// EVENT CODE //
	FB_AlarmCodeManager(
		bAlarm1			:= TON_BatteriesCharging.Q ,								//Batteries charging
		bAlarm2			:= TON_BatteriesDischarging.Q,								//Batteries discharging
		bAlarm3			:= FALSE,													//
		bAlarm4			:= FALSE,													//		
		bAlarm5			:= IN_CmdOpenDC,                                            // Open DC command
		bAlarm6			:= IN_CmdCloseDC,                                           // Close DC Command
		bAlarm7			:= FALSE,                                                   //
		bAlarm8			:= FALSE,                                                   //
		bAlarm9			:= FALSE,                                                   //
		bAlarm10		:= FALSE,                                                   //
		bAlarm11		:= FALSE,                                                   //
		bAlarm12		:= FALSE,                                                   //
		bAlarm13		:= FALSE,                                                   //
		bAlarm14		:= FALSE,                                                   //
		bAlarm15		:= FALSE,                                                   //
		wAlarmCode		=> MesDataExd.MesData.MesEventCode);


	FB_AlarmCodeManager(	
        bAlarm1			:= MesDataExd.MesChargeStatus= 1,  									// Charge Status  -  OFF
        bAlarm2			:= MesDataExd.MesChargeStatus= 2,  									// Charge Status  -  EMPTY
        bAlarm3			:= MesDataExd.MesChargeStatus= 3,  									// Charge Status  -  DISCHARGING
        bAlarm4			:= MesDataExd.MesChargeStatus= 4,  									// Charge Status  -  CHARGING
        bAlarm5			:= MesDataExd.MesChargeStatus= 5,  									// Charge Status  -  FULL
        bAlarm6			:= MesDataExd.MesChargeStatus= 6,  									// Charge Status  -  HOLDING
        bAlarm7			:= MesDataExd.MesChargeStatus= 7,  									// Charge Status  -  TESTING
		bAlarm8			:= FALSE,                                                   //
		bAlarm9			:= FALSE,                                                   //
		bAlarm10		:= FALSE,                                                   //
		bAlarm11		:= FALSE,                                                   //
		bAlarm12		:= FALSE,                                                   //
		bAlarm13		:= FALSE,                                                   //
		bAlarm14		:= FALSE,                                                   //
		bAlarm15		:= FALSE,                                                   //
		wAlarmCode		=> MesDataExd.MesChargeStatus);

		

	FB_AlarmCodeManager(	
        bAlarm1			:= MesIDState= 1,  				// State of the Battery Bank  -  DISCONNECTED
        bAlarm2			:= MesIDState= 2,  				// State of the Battery Bank  -  INITIALIZING
        bAlarm3			:= MesIDState= 3,  				// State of the Battery Bank  -  CONNECTED
        bAlarm4			:= MesIDState= 4,  				// State of the Battery Bank  -  STANDBY
        bAlarm5			:= MesIDState= 5,  				// State of the Battery Bank  -  SOC PROTECTION
        bAlarm6			:= MesIDState= 6,  				// State of the Battery Bank  -  SUSPENDING
        bAlarm7			:= MesIDState= 99,  			// State of the Battery Bank  -  FAULT
		bAlarm8			:= FALSE,                       //
		bAlarm9			:= FALSE,                       //
		bAlarm10		:= FALSE,                       //
		bAlarm11		:= FALSE,                       //
		bAlarm12		:= FALSE,                       //
		bAlarm13		:= FALSE,                       //
		bAlarm14		:= FALSE,                       //
		bAlarm15		:= FALSE,                       //
		wAlarmCode		=> MesDataExd.MesData.MesIDState
);
(*
	FB_AlarmCodeManager(	
        bAlarm1		:= MesData.MesEvt1.0,  			// Battery Event 1 -  COMMUNICATION_ERROR
        bAlarm2		:= MesData.MesEvt1.1,  			// Battery Event 1 -  OVER_TEMP_ALARM
        bAlarm3		:= MesData.MesEvt1.2,  			// Battery Event 1 -  OVER_TEMP_WARNING
        bAlarm4		:= MesData.MesEvt1.3,  			// Battery Event 1 -  UNDER_TEMP_ALARM
        bAlarm5		:= MesData.MesEvt1.4,  			// Battery Event 1 -  UNDER_TEMP_WARNING
        bAlarm6		:= MesData.MesEvt1.5,  			// Battery Event 1 -  OVER_CHARGE_CURRENT_ALARM
        bAlarm7		:= MesData.MesEvt1.6,  			// Battery Event 1 -  OVER_CHARGE_CURRENT_WARNING
        bAlarm8		:= MesData.MesEvt1.7,  			// Battery Event 1 -  OVER_DISCHARGE_CURRENT_ALARM
        bAlarm9		:= MesData.MesEvt1.8,  			// Battery Event 1 -  OVER_DISCHARGE_CURRENT_WARNING
        bAlarm10	:= MesData.MesEvt1.9,  			// Battery Event 1 -  OVER_VOLT_ALARM
        bAlarm11	:= MesData.MesEvt1.10,  		// Battery Event 1 -  OVER_VOLT_WARNING
        bAlarm12	:= MesData.MesEvt1.11,  		// Battery Event 1 -  UNDER_VOLT_ALARM
        bAlarm13	:= MesData.MesEvt1.12,  		// Battery Event 1 -  UNDER_VOLT_WARNING
        bAlarm14	:= MesData.MesEvt1.13,  		// Battery Event 1 -  UNDER_SOC_MIN_ALARM
        bAlarm15	:= MesData.MesEvt1.14,  		// Battery Event 1 -  UNDER_SOC_MIN_WARNING
		wAlarmCode	=> MesData.MesAlarmCode_MesEvt1_1
);

	FB_AlarmCodeManager(	
        bAlarm1		:= MesData.MesEvt1.15,  		// Battery Event 1 -  OVER_SOC_MAX_ALARM
        bAlarm2		:= MesData.MesEvt1.16,  		// Battery Event 1 -  OVER_SOC_MAX_WARNING
        bAlarm3		:= MesData.MesEvt1.17,  		// Battery Event 1 -  VOLTAGE_IMBALANCE_WARNING
        bAlarm4		:= MesData.MesEvt1.18,  		// Battery Event 1 -  TEMPERATURE_IMBALANCE_ALARM
        bAlarm5		:= MesData.MesEvt1.19,  		// Battery Event 1 -  TEMPERATURE_IMBALANCE_WARNING
        bAlarm6		:= MesData.MesEvt1.20,  		// Battery Event 1 -  CONTACTOR_ERROR
        bAlarm7		:= MesData.MesEvt1.21,  		// Battery Event 1 -  FAN_ERROR
        bAlarm8		:= MesData.MesEvt1.22,  		// Battery Event 1 -  GROUND_FAULT
        bAlarm9		:= MesData.MesEvt1.23,  		// Battery Event 1 -  OPEN_DOOR_ERROR
        bAlarm10	:= MesData.MesEvt1.24,  		// Battery Event 1 -  CURRENT_IMBALANCE_WARNING
        bAlarm11	:= MesData.MesEvt1.25,  		// Battery Event 1 -  OTHER_ALARM
        bAlarm12	:= MesData.MesEvt1.26,  		// Battery Event 1 -  OTHER_WARNING
        bAlarm13	:= MesData.MesEvt1.27,  		// Battery Event 1 -  RESERVED_1
        bAlarm14	:= MesData.MesEvt1.28,  		// Battery Event 1 -  CONFIGURATION_ALARM
        bAlarm15	:= MesData.MesEvt1.29,  		// Battery Event 1 -  CONFIGURATION_WARNING
		wAlarmCode	=> MesData.MesAlarmCode_MesEvt1_2
);

	FB_AlarmCodeManager(	
        bAlarm1			:= MesData.MesEvtVnd1.0,  		// Battery Vendor Event 1   -  Cell Over Voltage Warning   
        bAlarm2			:= MesData.MesEvtVnd1.1,  		// Battery Vendor Event 1   -  Cell Under Voltage Warning  
        bAlarm3			:= MesData.MesEvtVnd1.2,  		// Battery Vendor Event 1   -  Cell Voltage Imbalance      
        bAlarm4			:= MesData.MesEvtVnd1.3,  		// Battery Vendor Event 1   -  Cell Over Voltage Alarm     
        bAlarm5			:= MesData.MesEvtVnd1.4,  		// Battery Vendor Event 1   -  Cell Under Voltage Alarm    
        bAlarm6			:= MesData.MesEvtVnd1.5,  		// Battery Vendor Event 1   -  Cell Voltage Imbalance Alarm
        bAlarm7			:= MesData.MesEvtVnd1.6,  		// Battery Vendor Event 1   -  Cell Over Voltage Fault     
        bAlarm8			:= MesData.MesEvtVnd1.7,  		// Battery Vendor Event 1   -  Cell Under Voltage Fault    
        bAlarm9			:= MesData.MesEvtVnd1.8,  		// Battery Vendor Event 1   -  Cell Voltage Imbalance Fault
        bAlarm10		:= MesData.MesEvtVnd1.9,  		// Battery Vendor Event 1   -  Over Temperature Fault      
        bAlarm11		:= MesData.MesEvtVnd1.10,  	// Battery Vendor Event 1   -  Under Temperature Fault     
        bAlarm12		:= MesData.MesEvtVnd1.11,  	// Battery Vendor Event 1   -  Temperature Imbalance Fault 
        bAlarm13		:= MesData.MesEvtVnd1.12,  	// Battery Vendor Event 1   -  Over Voltage Fault          
        bAlarm14		:= MesData.MesEvtVnd1.13,  	// Battery Vendor Event 1   -  Under Voltage Fault         
        bAlarm15		:= MesData.MesEvtVnd1.14,  	// Battery Vendor Event 1   -  Over Charge Current Fault   
		wAlarmCode		=>MesData.MesAlarmCode_MesEvtVnd1_1
);

	FB_AlarmCodeManager(	
        bAlarm1			:= MesData.MesEvtVnd1.15,  	// Battery Vendor Event 1  -  Over Discharge Current Fault      
        bAlarm2			:= MesData.MesEvtVnd1.16,  	// Battery Vendor Event 1  -  String Connection Failure         
        bAlarm3			:= MesData.MesEvtVnd1.17,  	// Battery Vendor Event 1  -  RBMS to MBMS Communication Failure
        bAlarm4			:= MesData.MesEvtVnd1.18,  	// Battery Vendor Event 1  -  Temperature Sensor Failure       
        bAlarm5			:= MesData.MesEvtVnd1.19,  	// Battery Vendor Event 1  -  Main Relay Open Failure          
        bAlarm6			:= MesData.MesEvtVnd1.20,  	// Battery Vendor Event 1  -  Bus Voltage Imbalance             
        bAlarm7			:= MesData.MesEvtVnd1.21,  	// Battery Vendor Event 1  -  Fan Failure                       
        bAlarm8			:= MesData.MesEvtVnd1.22,  	// Battery Vendor Event 1  -  Voltage Sensor Failure            
        bAlarm9			:= MesData.MesEvtVnd1.23,  	// Battery Vendor Event 1  -  Insulation Detection Warning      
        bAlarm10		:= MesData.MesEvtVnd1.24,  	// Battery Vendor Event 1  -  Insulation Detection Fault        
		bAlarm11		:= FALSE,                                                   //
		bAlarm12		:= FALSE,                                                   //
		bAlarm13		:= FALSE,                                                   //
		bAlarm14		:= FALSE,                                                   //
		bAlarm15		:= FALSE,                                                   //
		wAlarmCode		=> MesData.MesAlarmCode_MesEvtVnd1_2
);
*)
END_METHOD

METHOD M_CP
//////////////////
//  Permanent conditions 
/////////////////

VAR 
	// Method local variables (reinitialized at each cycle) 
	
END_VAR


SUPER^.M_CP() ; 




Trig_Cmd_Read(CLK:=IN_CmdToggleRead);
Trig_Cmd_Write(CLK:=IN_CmdToggleWrite);
	
IF Trig_Cmd_Read.Q THEN
	IN_CmdToggleRead := FALSE;
	MesDataExd.MesData.MesCP_Read := NOT MesDataExd.MesData.MesCP_Read;
END_IF


IF Trig_Cmd_Write.Q THEN
	IN_CmdToggleWrite := FALSE;
	MesDataExd.MesData.MesCP_Write := NOT MesDataExd.MesData.MesCP_Write;
END_IF
END_METHOD

METHOD M_Evaluate : BOOL
VAR_INPUT
END_VAR
VAR
	KK : UINT;
	
END_VAR
MesDataExd.MesNbRackConnected := 0;
MesDataExd.MesData.MesEnomConnected := 0;
//MesDataExd.MesData.MesSoC_Max := MesDataExd.AX_RACK[1].MesSoC;
//MesDataExd.MesData.MesSoC_Min := MesDataExd.AX_RACK[1].MesSoC;

// Initialisation des valeurs min et max
//--------------------------------------------------------------------
MesDataExd.MesData.MesSoC_Max :=0;
MesDataExd.MesData.MesSoC_Min :=0;
MesDataExd.MesSoCConnected:=0;

FOR KK := 1 TO CstNbRack_BAT_G DO		
	IF MesDataExd.AX_RACK[KK].MesData.MesIDState = 5 THEN
		MesDataExd.MesData.MesSoC_Min:=MesDataExd.AX_RACK[KK].MesData.MesSoC;
		MesDataExd.MesData.MesSoC_Max:=MesDataExd.AX_RACK[KK].MesData.MesSoC;
	END_IF
END_FOR
//--------------------------------------------------------------------

FOR KK := 1 TO CstNbRack_BAT_G DO
		
	IF MesDataExd.AX_RACK[KK].MesData.MesIDState = 5 THEN
		IF MesDataExd.MesData.MesSoC_Min = 0 THEN
			MesDataExd.MesData.MesSoC_Min := MesDataExd.AX_RACK[KK].MesData.MesSoC;
		END_IF
		MesDataExd.MesData.MesSoC_Max := MAX(MesDataExd.MesData.MesSoC_Max, MesDataExd.AX_RACK[KK].MesData.MesSoC);
		MesDataExd.MesData.MesSoC_Min := MIN(MesDataExd.MesData.MesSoC_Min, MesDataExd.AX_RACK[KK].MesData.MesSoC);
	END_IF
	MesDataExd.MesNbRackConnected := MesDataExd.MesNbRackConnected + SEL(MesDataExd.AX_RACK[KK].MesData.MesIDState = 5, 0, 1);
	MesDataExd.MesData.MesEnomConnected := MesDataExd.MesData.MesEnomConnected + SEL(MesDataExd.AX_RACK[KK].MesData.MesIDState = 5, 0, ParamEnomRack) ;
	MesDataExd.MesSoCConnected := MesDataExd.MesSoCConnected + SEL(MesDataExd.AX_RACK[KK].MesData.MesIDState = 5, 0, MesDataExd.AX_RACK[KK].MesData.MesSoC);
END_FOR


	
	MesDataExd.MesSoCConnected := SEL(MesDataExd.MesNbRackConnected>1 , 0 , MesDataExd.MesSoCConnected / MesDataExd.MesNbRackConnected ) ;

	
	
	(* EN DOUBLE AVEC CODE PCS 
// Gestion des Start/Stop par SOC Low
	TRIG_SocOpenDC(clk := MesDataExd.MesData.MesState.0 AND NOT MesDataExd.MesData.MesState.4 AND (MesDataExd.MesUdcMin_Cell <= ParamVdcL OR MesDataExd.MesUdcMin_Cell >= ParamVdcH));
	IF TRIG_SocOpenDC.Q THEN
		MesDataExd.MesData.MesState.4 := TRUE;
	END_IF
	
	
	TRIG_SocOpenDc_Again(CLK := Time_Discharge_LowSoc > ParamTimeLowSocToRecharge);
	IF MesDataExd.MesData.MesState.0 AND MesDataExd.MesData.MesState.4 AND MesDataExd.MesData.MesPdc > 0 THEN
		Time_Discharge_LowSoc := Time_Discharge_LowSoc + TIME() - Time_Start_Discharge_LowSoc;
	ELSIF NOT MesDataExd.MesData.MesState.0 AND (NOT MesDataExd.MesData.MesState.4 OR Time_Discharge_LowSoc >= ParamTimeLowSocToRecharge) THEN
		Time_Discharge_LowSoc := T#0S;
	END_IF
	Time_Start_Discharge_LowSoc := TIME();
	
	TRIG_BackToNormalSoc(CLK := MesDataExd.MesData.MesState.4 AND MesDataExd.MesData.MesSoC >= ParamSocStop);
	IF TRIG_BackToNormalSoc.Q THEN
		MesDataExd.MesData.MesState.4 := 0;
	END_IF
*)
END_METHOD

METHOD M_Init
VAR 

END_VAR
END_METHOD

METHOD M_Read
//////////////////
//  Ici, la lecture est séparée en Modèles Sunspec : 802 est le modèle de base pour le MsBMS
// 803 est le modèle de base pour les strings : une partie fixe pour l'ensemble + partie variable par string
// 804 est le modèle de base pour les modules : une partie fixe par rack + partie variable par string 
/////////////////

VAR 
	// Method local variables (reinitialized at each cycle) 
	MW1 	: FB_MergeWordsToFloat ; 
	MW2		: FB_MergeWordsToUint;
	MW 		: FB_MergeWordsToDint;
	JJ			: DINT;
	KK			: DINT;
	LL			: DINT;
	MM			: DINT;
	MW_U	: FB_MergeWordsToUint ;

	IDState_UINT : UINT;
	IDAlarm			: UINT;
	ID_Evt1			: UINT;
	ID_Evt2			: UINT;
	ID_EvtVnd1		: UINT;
	ID_EvtVnd2		: UINT;
END_VAR


IF MesDataExd.MesData.MesCP_Read  THEN	
	ModbusRead802
	(
		pDestAddr 	:= ADR(MesBlock_802),
		sIPAddr 	:= ParamIpAddress,
		tTimeout 	:= ParamTimeout,
		nTcpPort 	:= 8694,
		nQuantity 	:= 64,
		nMBAddr 	:= StartAddr,
		cbLength 	:= SIZEOF(MesBlock_802),
		nUnitID		:= 1,
		ClockRead	:= ClockRead,
		ModbusReadAlarm => MesModbusReadAlarm[1] , 
		OUT_NbRead	=> NbRead
	);
	
	Cal_StartRead803_Fix := StartAddr + 64;
	ModbusRead803_Fix
	(
		pDestAddr 	:= ADR(MesBlock_803_Fix),
		sIPAddr 	:= ParamIpAddress,
		tTimeout 	:= ParamTimeout,
		nTcpPort 	:= 8694,
		nQuantity 	:= 28,
		nMBAddr 	:= Cal_StartRead803_Fix,
		cbLength 	:= SIZEOF(MesBlock_803_Fix),
		nUnitID		:= 1,
		ModbusReadAlarm => MesModbusReadAlarm[2] , 
		ClockRead	:= ClockRead
	);
	
	
	
	FOR KK := 1 TO ParamNbRacks DO
		
		ModbusRead803_Rep[KK]
		(
			pDestAddr 	:= ADR(MesBlock_803_Rep[KK]),
			sIPAddr 	:= ParamIpAddress,
			tTimeout 	:= ParamTimeout,
			nTcpPort 	:= 8694,
			nQuantity 	:= 32,
			nMBAddr 	:= Cal_StartRead803_Fix + 28 + DINT_TO_WORD(KK-1)*32,
			cbLength 	:= SIZEOF(MesBlock_803_Rep[KK]),
			nUnitID		:= 1,
			ModbusReadAlarm => MesModbusReadAlarmRacks[KK][1] , 
			ClockRead	:= ClockRead
		);	
	
	
		// Début du 804 = Début 803 fixe + nb 803 fix (=28) + nombre de strings * nombre registres dans 803 rep (=32)
		
		Cal_StartRead804_Fix := Cal_StartRead803_Fix + 28 + ParamNbRacks*32 ;
   		//Cal_StartRead804_Fix := 1218;
		
		ModbusRead804_Fix[KK]
		(
			pDestAddr 	:= ADR(MesBlock_804_Fix[KK]),
			sIPAddr 	:= ParamIpAddress,
			tTimeout 	:= ParamTimeout,
			nTcpPort 	:= 8694, //8694,
			nQuantity 	:= 46,
			nMBAddr 	:= Cal_StartRead804_Fix + DINT_TO_WORD(KK - 1)*(48),
			cbLength 	:= SIZEOF(MesBlock_804_Fix[KK]),
			nUnitID		:= 1,
			ModbusReadAlarm => MesModbusReadAlarmRacks[KK][2] , 
			ClockRead	:= ClockRead
		);
		
    
	END_FOR
	
	

// Attributions
	MesAHRtg_SF_802					:= EXPT(10, INT_TO_REAL( WORD_TO_INT(MesBlock_802[53])));
	MesWHRtg_SF_802					:= EXPT(10, INT_TO_REAL( WORD_TO_INT(MesBlock_802[54])));
	MesWChaDisChaMax_SF_802			:= EXPT(10, INT_TO_REAL( WORD_TO_INT(MesBlock_802[55])));
	MesDisChaRte_SF_802				:= EXPT(10, INT_TO_REAL( WORD_TO_INT(MesBlock_802[56])));
	MesSoC_SF_802					:= EXPT(10, INT_TO_REAL( WORD_TO_INT(MesBlock_802[57])));
	MesDoD_SF_802					:= EXPT(10, INT_TO_REAL( WORD_TO_INT(MesBlock_802[58])));
	MesSoH_SF_802					:= EXPT(10, INT_TO_REAL( WORD_TO_INT(MesBlock_802[59])));
	MesV_SF_802						:= EXPT(10, INT_TO_REAL( WORD_TO_INT(MesBlock_802[60])));
	MesCellV_SF_802					:= EXPT(10, INT_TO_REAL( WORD_TO_INT(MesBlock_802[61])));
	MesA_SF_802 					:= EXPT(10, INT_TO_REAL( WORD_TO_INT(MesBlock_802[62])));
	MesAMax_SF_802 					:= EXPT(10, INT_TO_REAL( WORD_TO_INT(MesBlock_802[63])));
	MesW_SF_802 					:= EXPT(10, INT_TO_REAL( WORD_TO_INT(MesBlock_802[64])));
	
	MesSoC_SF_803 	            	:= EXPT(10, INT_TO_REAL( WORD_TO_INT(MesBlock_803_Fix[27])));
	MesSoH_SF_803 	            	:= EXPT(10, INT_TO_REAL( WORD_TO_INT(MesBlock_803_Fix[26])));
	MesA_SF_803 	            	:= EXPT(10, INT_TO_REAL( WORD_TO_INT(MesBlock_803_Fix[25])));
	MesV_SF_803 	            	:= EXPT(10, INT_TO_REAL( WORD_TO_INT(MesBlock_803_Fix[28])));
	MesCellV_SF_803					:= EXPT(10, INT_TO_REAL( WORD_TO_INT(MesBlock_803_Fix[23]))); 
	MesModTmp_SF_803            	:= EXPT(10, INT_TO_REAL( WORD_TO_INT(MesBlock_803_Fix[24])));
	MesSoH_SF_803					:= EXPT(10, INT_TO_REAL( WORD_TO_INT(MesBlock_803_Fix[25])));
	
	MesDataExd.MesNbCycle 			:= WORD_TO_UINT(MesBlock_802[15]);
	MesChargeStatus 				:= WORD_TO_UINT(MesBlock_802[17]);
	MesDataExd.MesRemoteControl 	:= MesBlock_802[18]=0;
	MesDataExd.MesHeartBeat 		:= WORD_TO_UINT(mesblock_802[19]);
	MesDataExd.MesTypeBattery 		:= MesBlock_802[22];
	MesIDState 						:= WORD_TO_UINT(MesBlock_802[23]);
	MW_U(word_strong := MesBlock_802[27], word_weak := mesblock_802[28], VAR_OUT:= IDAlarm);
	MesDataExd.MesIDAlarm := UINT_TO_DWORD(IDAlarm); 
//	MW(WORD_STRONG:= MesBlock_802[27], SIGNED:=TRUE, FIX:=1 , SIZE:=1, VAR_OUT:=MesDataExd.MesData.MesUdc);
	
	MesDataExd.MesIDRack_UdcMax_Cell := WORD_TO_UINT(MesBlock_802[39]);
	MesDataexd.MesIDModule_UdcMax_Cell := WORD_TO_UINT(MesBlock_802[40]);
	MesDataExd.MesIDRack_UdcMin_Cell := WORD_TO_UINT(MesBlock_802[42]);
	MesDataexd.MesIDModule_UdcMin_Cell := WORD_TO_UINT(MesBlock_802[43]);
	

	
	IF MesA_SF_802 <> 0 THEN
		MW(WORD_STRONG := mesblock_802[45], signed := TRUE,	size := 1, fix := REAL_TO_INT(1/MesA_SF_802), var_out := MesDataExd.MesData.MesIdc);
	END_IF
	
	
	IF MesWChaDisChaMax_SF_802 <> 0 THEN
		MesDataExd.MesData.MesCPL		:=  WORD_TO_REAL(MesBlock_802[5])/MesWChaDisChaMax_SF_802;
		MesDataExd.MesData.MesDPL		:=  WORD_TO_REAL(MesBlock_802[6])/MesWChaDisChaMax_SF_802;
	END_IF
	
	
	IF MesSoC_SF_802 <> 0 THEN
		// SI aucun string connecté, le SoC passe à 65535
		IF MesDataExd.MesNbRackTot <> 0 THEN
			MesDataExd.MesData.MesSoC			:=  WORD_TO_REAL(MesBlock_802[12])*MesSoC_SF_802;
		ELSE
		    MesDataExd.MesData.MesSoC			:= 0;
		END_IF
	END_IF
	
	IF MesDoD_SF_802 <> 0 THEN
		MesDataExd.MesData.MesDoD :=  WORD_TO_REAL(MesBlock_802[13]) *MesDoD_SF_802;
	END_IF
	
	IF MesSoH_SF_802 <> 0 THEN
		MesDataExd.MesData.MesSoH :=  WORD_TO_REAL(MesBlock_802[14])*MesSoH_SF_802;
	END_IF
	
	IF MesV_SF_802 <> 0 THEN
		MesDataExd.MesData.MesUdc 		:=  WORD_TO_REAL(MesBlock_802[35])*MesV_SF_802;
		//MesDataExd.MesData.MesUdcMax 	:=  WORD_TO_REAL(MesBlock_802[36])*MesV_SF_802;
		//MesDataExd.MesData.MesUdcMin 	:=  WORD_TO_REAL(MesBlock_802[37])*MesV_SF_802;
	END_IF
	
	IF MesCellV_SF_802 <> 0 THEN
		MesDataExd.MesUdcMax_Cell :=  WORD_TO_REAL(MesBlock_802[38])*MesCellV_SF_802;
		MesDataexd.MesUdcMin_Cell :=  WORD_TO_REAL(MesBlock_802[41])*MesCellV_SF_802;
		//MesDataExd.MesData.MesUdc :=  WORD_TO_REAL(MesBlock_802[44])*MesCellV_SF_802;
	END_IF
	
	
	IF MesAMax_SF_802 <> 0 THEN
		MesDataExd.MesData.MesCCL :=  WORD_TO_REAL(MesBlock_802[46])*MesAMax_SF_802;
		MesDataExd.MesData.MesDCL :=  WORD_TO_REAL(MesBlock_802[47])*MesAMax_SF_802;
	END_IF
	
	IF MesW_SF_802 <> 0 THEN
		MW(WORD_STRONG := mesblock_802[48], size := 1, SIGNED := TRUE,fix := REAL_TO_INT(1/MesW_SF_802), var_out := MesDataExd.MesData.MesPdc);
	END_IF
	
	//MesDataExd.MesNbRackConnected	 	:= WORD_TO_UINT(MesBlock_803_Fix[3]);
	MesDataExd.MesNbRackTot 			:= WORD_TO_UINT(MesBlock_803_Fix[4]);
	
	MesDataExd.MesIDRack_TempMax_Module 	:= WORD_TO_UINT(MesBlock_803_Fix[6]);
	MesDataExd.MesIDModule_TempMax_Module 	:= WORD_TO_UINT(MesBlock_803_Fix[7]);
	MesDataExd.MesIDRack_TempMin_Module 	:= WORD_TO_UINT(MesBlock_803_Fix[9]);
	MesDataExd.MesIDModule_TempMin_Module 	:= WORD_TO_UINT(MesBlock_803_Fix[10]);
	
	MesDataExd.MesIDRack_UdcMax_Rack 		:= WORD_TO_UINT(MesBlock_803_Fix[13]);
	MesDataExd.MesIDRack_UdcMin_Rack 		:= WORD_TO_UINT(MesBlock_803_Fix[15]);
	
	MesDataExd.MesIDRack_Imax_Rack			:= WORD_TO_UINT(MesBlock_803_Fix[18]);
	MesDataExd.MesIDRack_Imin_Rack			:= WORD_TO_UINT(MesBlock_803_Fix[20]);
	
	MesDataExd.MesNbCellbalancing 			:= WORD_TO_UINT(MesBlock_803_Fix[22]);
	
	IF MesA_SF_803 <> 0 THEN
		MesDataExd.MesIdcmax_Rack			:= WORD_TO_REAL(MesBlock_803_Fix[17])*MesA_SF_803;
		MesDataExd.MesIdcMin_Rack			:= WORD_TO_REAL(MesBlock_803_Fix[19])*MesA_SF_803;
		MesDataExd.MesIdc_Rack				:= WORD_TO_REAL(MesBlock_803_Fix[21])*MesA_SF_803;
	END_IF
	
	IF MesV_SF_803 <> 0 THEN
		MesDataExd.MesUdcMax_Rack			:= WORD_TO_REAL(MesBlock_803_Fix[12])*MesV_SF_803;
		MesDataExd.MesUdcMin_Rack			:= WORD_TO_REAL(MesBlock_803_Fix[14])*MesV_SF_803;
		MesDataExd.MesUdc_Rack				:= WORD_TO_REAL(MesBlock_803_Fix[16])*MesV_SF_803;
	END_IF
	
	IF MesModTmp_SF_803 <> 0 THEN
		MesDataExd.MesTempMax_Module		:= WORD_TO_REAL(MesBlock_803_Fix[5])*mesmodtmp_sf_803;
		MesDataExd.MesTempMin_Module		:= WORD_TO_REAL(MesBlock_803_Fix[8])*mesmodtmp_sf_803;
		MesDataExd.MesTemp_Module			:= WORD_TO_REAL(MesBlock_803_Fix[11])*mesmodtmp_sf_803;
	END_IF
	
	MesSoC_SF_804 	            :=EXPT(10, INT_TO_REAL(WORD_TO_INT(MesBlock_804_Fix[1][39])));
	MesSoH_SF_804 	            :=EXPT(10, INT_TO_REAL( WORD_TO_INT(MesBlock_804_Fix[1][40])));
	MesDoD_SF_804 	            :=EXPT(10, INT_TO_REAL( WORD_TO_INT(MesBlock_804_Fix[1][41])));
	MesA_SF_804 	            :=EXPT(10, INT_TO_REAL( WORD_TO_INT(MesBlock_804_Fix[1][42])));
	MesV_SF_804 	            :=EXPT(10, INT_TO_REAL( WORD_TO_INT(MesBlock_804_Fix[1][43])));
	MesCellV_SF_804				:=EXPT(10, INT_TO_REAL( WORD_TO_INT(MesBlock_804_Fix[1][44]))); 
	MesModTmp_SF_804            :=EXPT(10, INT_TO_REAL( WORD_TO_INT(MesBlock_804_Fix[1][45])));
	
	FOR KK := 1 TO ParamNbRacks DO
		MesDataExd.AX_Rack[KK].MesData.MesNbModuleTot 			:= WORD_TO_UINT(MesBlock_804_Fix[KK][4]);
		MW2(word_strong := MesBlock_803_Rep[KK][20], word_weak := MesBlock_803_Rep[KK][19], VAR_OUT := IDState_UINT);
		MesDataExd.AX_Rack[KK].MesData.MesIDState := UINT_TO_DWORD(IDState_UINT);
		
		MesDataExd.AX_RACK[KK].MesData.MesIDConnectAlarm	 	:= MesBlock_804_Fix[KK][7];
		MesDataExd.AX_RACK[KK].MesData.MesNbCellbalancing	 	:= WORD_TO_UINT(MesBlock_804_Fix[KK][8]);
		IF MesSoC_SF_804 <> 0 THEN
			MesDataExd.AX_RACK[KK].MesData.MesSoC			:= WORD_TO_REAL(MesBlock_804_Fix[KK][9])*MesSoC_SF_804;
		END_IF
		IF MesDoD_SF_804 <> 0 THEN
			MesDataExd.AX_RACK[KK].MesData.MesDoD			:= WORD_TO_REAL(MesBlock_804_Fix[KK][10])*MesDoD_SF_804;
		END_IF
		IF MesSoH_SF_804 <> 0 THEN
			MesDataExd.AX_RACK[KK].MesData.MesSoH			:= WORD_TO_REAL(MesBlock_804_Fix[KK][11])*MesSoH_SF_804;
		END_IF
		//MW2(WORD_STRONG := MesBlock_804_Fix[KK][12], WORD_STRONG := MesBlock_804_Fix[KK][13], VAR_OUT := MesDataExd.AX_Rack[KK].MesNCyc);
		
		IF MesA_SF_804 <> 0 THEN
		
			xTestWord:=INT_TO_WORD(xTestInt); // Kore Power 
			xTestReal			:=  INT_TO_REAL(WORD_TO_INT(xTestWord))*MesA_SF_804;
			xTestReal1			:=  WORD_TO_REAL(xTestWord)*MesA_SF_804;
		
	
			MesDataExd.AX_RACK[KK].MesData.MesIdc			:=  INT_TO_REAL(WORD_TO_INT(MesBlock_804_Fix[KK][14]))*MesA_SF_804;
		END_IF                                                                            
		IF MesV_SF_804 <> 0 THEN                                                          
			MesDataExd.AX_RACK[KK].MesData.MesUdc			:=  WORD_TO_REAL(MesBlock_804_Fix[KK][15])*MesV_SF_804;
		END_IF
		
		IF MesCellV_SF_804 <> 0 AND MesCellV_SF_804 < 65535 THEN
			MesDataExd.AX_RACK[KK].MesData.MesUdcMax_Cell	:= WORD_TO_REAL(MesBlock_804_Fix[KK][16])*MesCellV_SF_804;
			MesDataExd.AX_RACK[KK].MesData.MesUdcMin_Cell	:= WORD_TO_REAL(MesBlock_804_Fix[KK][18])*MesCellV_SF_804;
			MesDataExd.AX_RACK[KK].MesData.MesUdc_Cell		:= WORD_TO_REAL(MesBlock_804_Fix[KK][20])*MesCellV_SF_804;
		END_IF

		MesDataExd.AX_RACK[KK].MesData.MesIDModule_UdcMax_Cell	:= WORD_TO_UINT(MesBlock_804_Fix[KK][17]);
		MesDataExd.AX_RACK[KK].MesData.MesIDModule_UdcMin_Cell	:= WORD_TO_UINT(MesBlock_804_Fix[KK][19]);
		
		IF MesModTmp_SF_804 <> 0 THEN
			MesDataExd.AX_RACK[KK].MesData.MesTempMax_Module	:= WORD_TO_REAL(MesBlock_804_Fix[KK][21])*MesModTmp_SF_804;
			MesDataExd.AX_Rack[KK].MesData.MesTempMin_Module	:= WORD_TO_REAL(MesBlock_804_Fix[KK][23])*MesModTmp_SF_804;
			MesDataExd.AX_Rack[KK].MesData.MesTemp_Module		:= WORD_TO_REAL(MesBlock_804_Fix[KK][25])*MesModTmp_SF_804;
		END_IF			
		
		MesDataExd.AX_Rack[KK].MesData.MesIDModule_TempMax_Module		:= WORD_TO_UINT(MesBlock_804_Fix[KK][22]);
		MesDataExd.AX_Rack[KK].MesData.MesIDModule_TempMin_Module		:= WORD_TO_UINT(MesBlock_804_Fix[KK][24]);
		MesDataExd.AX_Rack[KK].MesData.MesIDState_DCSwitch				:= MesBlock_804_Fix[KK][(LL-1)*3 + 27];
		MW2(word_strong := MesBlock_804_Fix[KK][29], word_weak := MesBlock_804_Fix[KK][30], VAR_OUT := ID_Evt1);
		MesDataExd.AX_RACK[KK].MesData.MesIDAlarm := UINT_TO_DWORD(ID_Evt1);
		
		MW2(word_strong := MesBlock_804_Fix[KK][33], word_weak := MesBlock_804_Fix[KK][34], VAR_OUT := ID_EvtVnd1);
		MesDataExd.AX_RACK[KK].MesData.MesIDAlarm_Vendor1 := UINT_TO_DWORD(ID_EvtVnd1);

	END_FOR
END_IF

SUPER^.M_Read();
END_METHOD

METHOD M_StartStop
//////////////////
//  Start or stop BBMS via CAN bus   
/////////////////

VAR 
	// Method local variables (reinitialized at each cycle) 

END_VAR

SUPER^.M_StartStop();
END_METHOD

METHOD M_StateManager
//////////////////
// Detect which is the state of the PCS system . 
/////////////////

VAR 
	// Method local variables (reinitialized at each cycle) 

	
END_VAR



MesDataExd.MesData.MesState.0 := MesDataExd.MesNbRackConnected = 0 ;
MesDataExd.MesData.MesState.1 :=   MesDataExd.MesNbRackConnected > 0 ;
END_METHOD

METHOD M_Write
VAR_INPUT
END_VAR
VAR
	InputAddr: WORD;
	RTCWord: ARRAY[1..6] OF BYTE;
	TriggerRTC: BOOL;

	MBWr: INT;
	

END_VAR
Trig_CmdCloseDC(CLK := Xtest);//IN_CmdCloseDC);


 //Trig_CmdOpenDC(CLK :=IN_CmdOpenDC);
IF Trig_CmdCloseDC.Q THEN
	IN_CmdCloseDC := FALSE;
	AX_Cmd[1] := 16#0001;
END_IF
IF Trig_CmdOpenDC.Q THEN
	IN_CmdOpenDC := FALSE;
	AX_Cmd[1] := 16#0002;
END_IF

AX_ModbusWrite[1]	// Close / Open DC 
(
	InputWord	:= AX_Cmd[1],
	sIPAddr 	:= ParamIpAddress,
	tTimeout 	:= ParamTimeout,
	nTCPport 	:= ParamTcpPort,
	nMBAddr 	:= 152,
	nUnitID 	:= ParamUnitID,
	WriteCmd 	:= MesDataExd.Mesdata.MesCP_Write AND (Trig_CmdOpenDC.Q OR Trig_CmdCloseDC.Q),
	ModbusWriteAlarm => AX_bAlarmWrite[1],
	ErrorId		=> AX_uAlarmWrite[1]
);

Trig_CmdReset(CLK := IN_CmdReset);
IF Trig_CmdReset.Q THEN			// lacth the fault date of events. WE HAVE TO CHECK FIRST THE FAULT BEFORE DOING IT/ 
	IN_CmdReset := FALSE;
END_IF

AX_ModbusWrite[2]	// Reset 
(
	InputWord	:= 1,
	sIPAddr 	:= ParamIpAddress,
	tTimeout 	:= ParamTimeout,
	nTCPport 	:= ParamTcpPort,
	nMBAddr 	:= 89,
	nUnitID 	:= ParamUnitID,
	WriteCmd 	:= Trig_CmdReset.Q AND MesDataExd.Mesdata.MesCP_Write,
	ModbusWriteAlarm => AX_bAlarmWrite[2],
	ErrorId		=> AX_uAlarmWrite[2]
);

//Trig_Watchdog(CLK := CalLocalTimeStruct.wMilliseconds < 500 );	// watchdog every 5 seconds . 
//
//AX_ModbusWrite[3]	// Heartbeat 
//(
//	InputWord	:= CalLocalTimeStruct.wSecond,
//	sIPAddr 	:= ParamIpAddress,
//	tTimeout 	:= ParamTimeout,
//	nTCPport 	:= ParamTcpPort,
//	nMBAddr 	:= 20,
//	nUnitID 	:= ParamUnitID,
//	WriteCmd 	:= Trig_Watchdog.Q AND MesDataExd.Mesdata.MesCP_Write,
//	ModbusWriteAlarm => AX_bAlarmWrite[3],
//	ErrorId		=> AX_uAlarmWrite[3]
//);
END_METHOD

END_FUNCTION_BLOCK

// ---- 01_Equipement_Library/Batteries/FB_BAT_Saft.TcPOU
FUNCTION_BLOCK FB_BAT_Saft EXTENDS FB_BAT_Base
// SAMSUNG System BMS P3
VAR_INPUT PERSISTENT
		ParamIpAddress 					: STRING 	:='192.168.1.51' ; 
		ParamUnitID						: BYTE  	:= 1 ; 
		ParamTcpPort					: UINT 		:= 502;
		ParamReadAlarmTime				: TIME 		:= T#1M30S;
		ParamReadWarningTime			: TIME		:= T#30S;
		ParamNbModule					: BYTE		:=24  ; // Nb of modules per strings .
 		ParamNbCells					: BYTE		:=16  ; // Nb of Cells per modules .
		ParamNbReadAtOnce				: BYTE		:=10 ; // Number of racks read at the same time . 
		ParamClockReadRack_Delay		: TIME 		:= T#500MS ; 			// Delay after bbms read and before rack read
		ParamEnom_Rack					: REAL 		:= 97;
END_VAR

VAR_INPUT
	
		IN_CmdOpenDC					: BOOL;
		IN_CmdCloseDC 					: BOOL;
		
		
			MesDataExd				: BAT_SAFT ; 
		
END_VAR

VAR_OUTPUT
	//Child objects
		
END_VAR

VAR
	//M_ALARMMANAGEMENT VARIABLES//
	
		MesRackAlarmCode				: WORD ;
		MesRackAlarmCode2				: WORD ;
		MesRackWarningCode				: WORD ;
		MesRackWarningCode2				: WORD ; 
		TON_BatteriesCharging			: TON ;
		TON_BatteriesDischarging		: TON ;
		
		AX_AlarmWords						: ARRAY[1..75] OF ST_ValuesAlarms;
		AX_AlarmWords_Null					: ARRAY[1..75] OF ST_ValuesAlarms;
		NumAlarmsActive						: UINT;
		
		
		TON_Heartbit						: TON ; 
		CalHeartbit_old						: UINT;
	//M_READ VARIABLES//
	

	
		ModbusRead						: ARRAY[1..3] OF FB_ModbusReadInputRegs  ; 
		ModbusReadBMS					: ARRAY[1..CstNbBAT_ESS_G] OF FB_ModbusReadInputRegs  ; 
		ModbusReadrack					: ARRAY[1..CstNbRack_BAT_G] OF FB_ModbusReadInputRegs ; 
		ModbusReadmodule		        : ARRAY[1..CstNbModule_Rack_G] OF FB_ModbusReadInputRegs ; 

             			
		MesBlock1_Temp					: ARRAY[1..3] OF ARRAY[0..123] OF WORD ; 	
		MesBlockBMS_Temp				: ARRAY[1..CstNbBAT_ESS_G] OF ARRAY[0..123]  OF WORD ; 
		MesBlockRack_Temp				: ARRAY[1..CstNbRack_BAT_G] OF ARRAY[0..119] OF WORD ; 
		MesBlockModule_Temp				: ARRAY[1..CstNbModule_Rack_G] OF ARRAY[0..123]  OF WORD ; 
		
		
		
		MesModbusReadAlarm				: ARRAY[1..3] OF BOOL;	
		MesModbusReadAlarmID			: ARRAY[1..3] OF UDINT;
		MesModbusReadAlarmRack			: ARRAY[1..CstNbRack_BAT_G] OF BOOL;	
		MesModbusReadAlarmIDRack		: ARRAY[1..CstNbRack_BAT_G] OF UDINT;		
		MesModbusReadAlarmModule		: ARRAY[1..CstNbModule_Rack_G] OF BOOL;	
		MesModbusReadAlarmIDModule		: ARRAY[1..CstNbModule_Rack_G] OF UDINT;	
		

		CTU_ClockRead								: CTU ; 
		TON_ClockRead					: TON;
	
	//M_WRITE VARIABLES //
		AX_Cmd					AT%Q*	: ARRAY[1..3] OF WORD;
		AX_Cmd_Old						: ARRAY[1..3] OF WORD;
		AX_ModbusWrite					: ARRAY[1..3] OF FB_ModbusWriteSingleRegister;
		A1_ModbusWriteRTC				: FB_ModbusWrite ; 
		
		Trig_Watchdog					: R_TRIG;
		Trig_CmdOpenDC					: R_TRIG;
		Trig_CmdCloseDC					: R_TRIG;
		Trig_CmdReset					: R_TRIG;
		
		RS_OpenClose					: RS;

	//M_STATEMANAGER VARIABLES//
	
	//M_INIT VARIABLES //
	
	//M_EVALUATE VARIABLES //
		Trig_NewDay						: R_TRIG;
		Trig_Second						: R_TRIG;
		E_Throughput_Integrate			: FB_Integrate;
	//M_EXECUTE VARIABLES//
		AX_DFV 							: ARRAY[1..13] OF FB_DetectFixedValue;	
		AX_FV							: ARRAY[1..13] OF UINT;
		Counter							: INT ; 
		CmdReset_L						: BOOL;
END_VAR

METHOD M_AlarmManagement
//////////////////
//  Battery Area  Alarm Management 
/////////////////

VAR 
	// Method local variables (reinitialized at each cycle) 
	FB_AlarmCodeManager 		: FB_AlarmCodeManager ; 
                            	
	KK							: UINT;				// For Loop 
	LL							: UINT;
	                        	
	ComWarning					: BOOL;				// Aggregated communication warning
	ComAlarm					: BOOL;				// Aggregated communication Alarm
	CalLOCRBMS					: BOOL;				// Lost of Communication (LOC) between BBMS and RBMS . 
	
	CalRackWarningSynthesis		: BOOL;
	CalRackAlarmSynthesis		: BOOL;

	MesSyntheseAlarmStatus		: WORD;
	MesNbMots					: UINT;
	WordTest					: WORD;
	ID_Journal					: UINT;
	
	

	
	
END_VAR
(*
TON_ComWarning( in := MesModbusReadAlarm OR MesModbusReadAlarm2[1] OR MesModbusReadAlarm2[2] OR MesModbusReadAlarm2[3] OR MesModbusReadAlarm2[4] OR MesModbusReadAlarm2[5] OR MesModbusReadAlarm2[6] OR MesModbusReadAlarm2[7], PT := ParamReadWarningTime);
TON_ComAlarm(IN:=  MesModbusReadAlarm AND MesModbusReadAlarm2[1] AND MesModbusReadAlarm2[2]AND MesModbusReadAlarm2[3]AND MesModbusReadAlarm2[4]AND MesModbusReadAlarm2[5]AND MesModbusReadAlarm2[6]AND MesModbusReadAlarm2[7], PT := ParamReadAlarmTime);
MesComWarning := TON_ComWarning.Q;


TON_Heartbit( IN:= MesDataExd.MesData.MesHeartBeat= CalHeartbit_old , PT:= T#3S ) ; 


IF MesDataExd.MesData.MesHeartBeat<> CalHeartbit_old THEN 
	CalHeartbit_old := MesDataExd.MesData.MesHeartBeat ; 
END_IF 

MesDataExd.MesDataExd.MesData.MesComAlarm := TON_ComAlarm.Q OR TON_Heartbit.Q;		// IL FAUT ARRETER LE SPCS EN MOINS DE 5 SEC SI PERTE DU WATCHDOG 


	
// ALARM CODE //
	FB_AlarmCodeManager(	
		bAlarm1			:= MesDataExd.MesData.MesComAlarm, 									// Com alarm
		bAlarm2			:= AX_DFV[13].OUT_bStatic,									// Watchdog alarm
		bAlarm3			:= MesDataExd.MesRackProtection1 >0 ,  						// Rack Protection Synthesis  1                    
		bAlarm4			:= MesDataExd.MesRackProtection2 >0  ,  						// Rack Protection Synthesis  2                        
		bAlarm5			:= MesDataExd.MesRackStringProtection1 >0 , 					// RackStringProtection Synthesis 1               
		bAlarm6			:= MesDataExd.MesRackStringProtection2 >0 , 					// RackStringProtection Synthesis 2
		bAlarm7			:= MesDataExd.MesRackStringProtection3 >0  , 					// RackStringProtection Synthesis 3   
		bAlarm8			:= MesDataExd.MesRackStringProtection4 >0  , 					// RackStringProtection Synthesis 4   
		bAlarm9			:= MesDataExd.MesAlarm1 >0 , 				  					// System Alarm 1               
		bAlarm10		:= MesDataExd.MesAlarm2 >0 , 	 								// System Alarm 2               
		bAlarm11		:= FALSE , 													//  						                
		bAlarm12		:= FALSE , 													//  						                
		bAlarm13		:= FALSE , 													//  						                 
		bAlarm14		:= FALSE , 													//  						                 
		bAlarm15		:= FALSE , 													//  						
		wAlarmCode		=>MesDataExd.MesData.MesAlarmCode);


// WARNING CODE //
	FB_AlarmCodeManager(	
		bAlarm1			:= MesComWarning, 											// Communication warning 
		bAlarm2			:= MesDataExd.MesData.MesRackAlarm1 >0,								// Rack Warning Syntesis 1                 
		bAlarm3			:= MesDataExd.MesData.MesRackAlarm2 >0,								// Rack Warning Syntesis 2                  
		bAlarm4			:= MesDataExd.MesData.MesRackStringAlarm1 >0 ,  						// Rack String Warning Synthesis 1                    
		bAlarm5			:= MesDataExd.MesData.MesRackStringAlarm2 >0,  						// Rack String Warning Synthesis 2                    
		bAlarm6			:= MesDataExd.MesData.MesRackStringAlarm3 >0,  						// Rack String Warning Synthesis 3                    
		bAlarm7			:= MesDataExd.MesData.MesRackStringAlarm4 >0,   						// Rack String Warning Synthesis 4                    
		bAlarm8			:= FALSE,   												//         
		bAlarm9			:= FALSE,   												//         
		bAlarm10		:= FALSE,   												//         
		bAlarm11		:= FALSE,   												//         
		bAlarm12		:= FALSE,   												//         
		bAlarm13		:= FALSE,  													//         
		bAlarm14		:= FALSE,  													//         
		bAlarm15		:= FALSE,	    											// 
		wAlarmCode		=>MesDataExd.MesData.MesWarningCode);          
		


TON_BatteriesCharging(IN := MesDataExd.MesData.MesSystemMode.15, PT := T#30S);
TON_BatteriesDischarging(IN := MesDataExd.MesData.MesSystemMode.14, PT := T#30S);


// EVENT CODE //
	FB_AlarmCodeManager(
		bAlarm1			:= TON_BatteriesCharging.Q ,								//Batteries charging
		bAlarm2			:= TON_BatteriesDischarging.Q,								//Batteries discharging
		bAlarm3			:= FALSE,													//
		bAlarm4			:= FALSE,													//		
		bAlarm5			:= IN_CmdOpenDC,                                            // Open DC command
		bAlarm6			:= IN_CmdCloseDC,                                           // Close DC Command
		bAlarm7			:= FALSE,                                                   //
		bAlarm8			:= FALSE,                                                   //
		bAlarm9			:= FALSE,                                                   //
		bAlarm10		:= FALSE,                                                   //
		bAlarm11		:= FALSE,                                                   //
		bAlarm12		:= FALSE,                                                   //
		bAlarm13		:= FALSE,                                                   //
		bAlarm14		:= FALSE,                                                   //
		bAlarm15		:= FALSE,                                                   //
		wAlarmCode		=>MesDataExd.MesData.MesEventCode);
*)
END_METHOD

METHOD M_CP
//////////////////
//  Permanent conditions 
/////////////////

VAR 
	// Method local variables (reinitialized at each cycle) 
	
END_VAR


SUPER^.M_CP() ; 




Trig_Cmd_Read(CLK:=IN_CmdToggleRead);
Trig_Cmd_Write(CLK:=IN_CmdToggleWrite);
	
IF Trig_Cmd_Read.Q THEN
	IN_CmdToggleRead := FALSE;
	MesDataExd.MesData.MesCP_Read := NOT MesDataExd.MesData.MesCP_Read;
END_IF


IF Trig_Cmd_Write.Q THEN
	IN_CmdToggleWrite := FALSE;
	MesDataExd.MesData.MesCP_Write := NOT MesDataExd.MesData.MesCP_Write;
END_IF
END_METHOD

METHOD M_Evaluate : BOOL
VAR_INPUT
END_VAR
VAR
	KK : UINT;
	MinVdc : REAL;
	MaxVdc : REAL;
//	MinVdcRackId : UINT;
//	MaxVdcRackId : UINT;
//	MinVdcModuleId : UINT;
//	MaxVdcModuleId : UINT;	
	JJ: INT;
	Temp_Energy: REAL;
END_VAR

//
////Watchdog fixed value :
//	AX_DFV[13]
//	(
//		IN_Addr := ADR(MesDataExd.MesHeartBeat),
//		IN_EmptyStruct := ADR(AX_DFV[13]),
//		IN_Size := SIZEOF(MesDataExd.MesHeartBeat),
//		IN_Duration := ParamTimeWatchdog
//	);


SUPER^.M_Evaluate();
END_METHOD

METHOD M_Init
VAR 

END_VAR
END_METHOD

METHOD M_Read
//////////////////
//  Read CAN 2.0B Variables for racks and BBMS .  
/////////////////

VAR 
	// Method local variables (reinitialized at each cycle) 
	MW 	: FB_MergeWordsToDint ; 
	MW_U	: FB_MergeWordsToUint ;
	
	AX_Addr		: ARRAY[1..3] OF UINT := [ 40071, 40135 ];
	AX_Qty		: ARRAY[1..3] OF UINT := [	112		, 35	,97	];
	LL			: INT;
	KK			: BYTE;
	CalRackNb	: INT;
	JJ			: BYTE;

	CalRegisterBaseModel			: UINT;
	CalRegisterBatModel				: UINT;
	CalRegisterBSSModel				: UINT;
	CalRegisterStringModel			: UINT;
	CalRegisterModuleModel			: UINT;
	CalBatModelQty					: UINT;
	CalStringModelQty				: UINT;
	CalModuleModelQty				: UINT;
	CalBaseModelQty					: UINT;
	CalBSSModelQty					: UINT ; 
	
	FF: UINT;
END_VAR

// CP-Read / Write 


// System BMS 
IF MesDataExd.MesData.MesCP_Read  THEN	
	// 802 et 803 et BSS
	CalBaseModelQty		:= 62 ;
	
	CalBatModelQty		:= 26 + (ParamNbRacks * 32) ; 
	CalStringModelQty 	:= 46 + (ParamNbModule* 16)  ; 
	CalModuleModelQty 	:= 42 + (ParamNbCells * 4) ; 
	CalBSSModelQty		:= 50 ; 
	
	CalRegisterBaseModel := 40071 ; 
	CalRegisterBatModel := 40135 ; 

	CalRegisterStringModel :=  CalRegisterBatModel + CalBatModelQty + 2; 
	CalRegisterModuleModel := CalRegisterStringModel +  (CalStringModelQty + 2)* ParamNbRacks ; 
	CalRegisterBSSModel := CalRegisterModuleModel +   (CalModuleModelQty +2) * ParamNbRacks* ParamNbModule  ; 
	
	// 802
	ModbusRead[1]
	(
		pDestAddr 		:= ADR(MesBlock1_Temp[1]),		sIPAddr 		:= ParamIpAddress,			tTimeout 		:= ParamTimeout,
		nTcpPort 		:= ParamTcpPort,				nQuantity 		:= CalBaseModelQty,				nMBAddr 		:= CalRegisterBaseModel,				
		cbLength 		:= SIZEOF(MesBlock1_Temp[1]),	nUnitID 		:= ParamUnitID,				ClockRead 		:= Clockread AND  MesDataExd.MesData.MesCP_Read,
		Reset 			:= IN_CmdReset,					ModbusReadAlarm => MesModbusReadAlarm[1],	ErrorId 		=> MesModbusReadAlarmID[1]
	);
	
	//803
	ModbusRead[2]
	(
		pDestAddr 		:= ADR(MesBlock1_Temp[2]),		sIPAddr 		:= ParamIpAddress,			tTimeout 		:= ParamTimeout,
		nTcpPort 		:= ParamTcpPort,				nQuantity 		:= CalBatModelQty,				nMBAddr 		:= CalRegisterBatModel,				
		cbLength 		:= SIZEOF(MesBlock1_Temp[2]),	nUnitID 		:= ParamUnitID,				ClockRead 		:= Clockread AND  MesDataExd.MesData.MesCP_Read,
		Reset 			:= IN_CmdReset,					ModbusReadAlarm => MesModbusReadAlarm[2],	ErrorId 		=> MesModbusReadAlarmID[2]
	);	
	
	
	
	// BSS
	ModbusRead[3]
	(
		pDestAddr 		:= ADR(MesBlock1_Temp[3]),		sIPAddr 		:= ParamIpAddress,			tTimeout 		:= ParamTimeout,
		nTcpPort 		:= ParamTcpPort,				nQuantity 		:= CalBSSModelQty,				nMBAddr 		:= CalRegisterBSSModel,				
		cbLength 		:= SIZEOF(MesBlock1_Temp[3]),	nUnitID 		:= ParamUnitID,				ClockRead 		:= Clockread AND  MesDataExd.MesData.MesCP_Read,
		Reset 			:= IN_CmdReset,					ModbusReadAlarm => MesModbusReadAlarm[3],	ErrorId 		=> MesModbusReadAlarmID[3]
	);		
	
	

	// MW() 
	
	MW(WORD_STRONG:= MesBlock1_Temp[1][ 1], SIGNED:=FALSE, FIX:=0 , SIZE:=1, VAR_OUT:=MesDataExd.MesData.MesChargeNom);
	MW(WORD_STRONG:= MesBlock1_Temp[1][ 2], SIGNED:=FALSE, FIX:=0 , SIZE:=1, VAR_OUT:=MesDataExd.MesData.MesEnom);
	MW(WORD_STRONG:= MesBlock1_Temp[1][ 3], SIGNED:=FALSE, FIX:=0 , SIZE:=1, VAR_OUT:=MesDataExd.MesData.MesPchargeNom);
	MW(WORD_STRONG:= MesBlock1_Temp[1][ 4], SIGNED:=FALSE, FIX:=0 , SIZE:=1, VAR_OUT:=MesDataExd.MesData.MesPDischargeNom);
	//MW(WORD_STRONG:= MesBlock1_Temp[1][ 5], SIGNED:=FALSE, FIX:=0 , SIZE:=1, VAR_OUT:=);
	//MW(WORD_STRONG:= MesBlock1_Temp[1][ 6], SIGNED:=FALSE, FIX:=0 , SIZE:=1, VAR_OUT:=);
	//MW(WORD_STRONG:= MesBlock1_Temp[1][ 7], SIGNED:=FALSE, FIX:=0 , SIZE:=1, VAR_OUT:=);
	//MW(WORD_STRONG:= MesBlock1_Temp[1][ 1], SIGNED:=FALSE, FIX:=0 , SIZE:=1, VAR_OUT:=);
	//MW(WORD_STRONG:= MesBlock1_Temp[1][ 1], SIGNED:=FALSE, FIX:=0 , SIZE:=1, VAR_OUT:=);
	MW(WORD_STRONG:= MesBlock1_Temp[1][ 10], SIGNED:=FALSE, FIX:=1 , SIZE:=1, VAR_OUT:=MesDataExd.MesData.MesSoC);
	//MW(WORD_STRONG:= MesBlock1_Temp[1][ 11], SIGNED:=FALSE, FIX:=1 , SIZE:=1, VAR_OUT:=MesDataExd.MesData.MesDoD);
	MW(WORD_STRONG:= MesBlock1_Temp[1][ 12], SIGNED:=FALSE, FIX:=0 , SIZE:=1, VAR_OUT:=MesDataExd.MesData.MesSoH);
	//MW(WORD_STRONG:= MesBlock1_Temp[1][ 1], SIGNED:=FALSE, FIX:=0 , SIZE:=1, VAR_OUT:=);
	//MW(WORD_STRONG:= MesBlock1_Temp[1][ 1], SIGNED:=FALSE, FIX:=0 , SIZE:=1, VAR_OUT:=);
	MesDataExd.MesData.MesID_ControlMode:=MesBlock1_Temp[1][16];
	MesDataExd.MesData.MesHeartbit:=MesBlock1_Temp[1][17];
	//MW(WORD_STRONG:= MesBlock1_Temp[1][ 18], SIGNED:=FALSE, FIX:=0 , SIZE:=1, VAR_OUT:=);
	//MW(WORD_STRONG:= MesBlock1_Temp[1][ 19], SIGNED:=FALSE, FIX:=0 , SIZE:=1, VAR_OUT:=);
	MesDataExd.MesData.MesID_BatType:=MesBlock1_Temp[1][20];
	MesDataExd.MesData.MesIDState:=MesBlock1_Temp[1][21];
	//MW(WORD_STRONG:= MesBlock1_Temp[1][ 1], SIGNED:=FALSE, FIX:=0 , SIZE:=1, VAR_OUT:=);
	//MW(WORD_STRONG:= MesBlock1_Temp[1][ 1], Word_WEAK:= MesBlock1_Temp[1][2], SIGNED:=FALSE, FIX:=0 , SIZE:=2, VAR_OUT:=);
	MW_U(WORD_STRONG:= MesBlock1_Temp[1][ 25], Word_WEAK:= MesBlock1_Temp[1][26], VAR_OUT:=MesDataExd.MesData.MesIDAlarm);
	//MW(WORD_STRONG:= MesBlock1_Temp[1][ 1], Word_WEAK:= MesBlock1_Temp[1][2], SIGNED:=FALSE, FIX:=0 , SIZE:=2, VAR_OUT:=);
	MW_U(WORD_STRONG:= MesBlock1_Temp[1][ 29], Word_WEAK:= MesBlock1_Temp[1][30], VAR_OUT:=MesDataExd.MesData.MesIDAlarm_Vendor1);
	MW_U(WORD_STRONG:= MesBlock1_Temp[1][ 31], Word_WEAK:= MesBlock1_Temp[1][32], VAR_OUT:=MesDataExd.MesData.MesIDAlarm_Vendor2);
	MW(WORD_STRONG:= MesBlock1_Temp[1][ 33], SIGNED:=FALSE, FIX:=1 , SIZE:=1, VAR_OUT:=MesDataExd.MesData.MesUdc);
	//MW(WORD_STRONG:= MesBlock1_Temp[1][ 34], SIGNED:=FALSE, FIX:=1 , SIZE:=1, VAR_OUT:=);
	//MW(WORD_STRONG:= MesBlock1_Temp[1][ 35], SIGNED:=FALSE, FIX:=1 , SIZE:=1, VAR_OUT:=);
	MW(WORD_STRONG:= MesBlock1_Temp[1][ 36], SIGNED:=FALSE, FIX:=3 , SIZE:=1, VAR_OUT:=MesDataExd.MesData.MesUdcMax_Cell);
	MesDataExd.MesData.MesIDRack_UdcMax_Cell:=MesBlock1_Temp[1][37];
	MesDataExd.MesData.MesIDModule_UdcMax_Cell:=MesBlock1_Temp[1][38];
	MW(WORD_STRONG:= MesBlock1_Temp[1][ 39], SIGNED:=FALSE, FIX:=3 , SIZE:=1, VAR_OUT:=MesDataExd.MesData.MesUdcMin_Cell);
	MesDataExd.MesData.MesIDRack_UdcMin_Cell:=MesBlock1_Temp[1][40];
	MesDataExd.MesData.MesIDModule_UdcMin_Cell:=MesBlock1_Temp[1][41];
	//MW(WORD_STRONG:= MesBlock1_Temp[1][ 42], SIGNED:=FALSE, FIX:=3 , SIZE:=1, VAR_OUT:=);
	MW(WORD_STRONG:= MesBlock1_Temp[1][ 43], SIGNED:=TRUE, FIX:=0 , SIZE:=1, VAR_OUT:=MesDataExd.MesData.MesIdc);
	MW(WORD_STRONG:= MesBlock1_Temp[1][ 44], SIGNED:=FALSE, FIX:=0 , SIZE:=1, VAR_OUT:=MesDataExd.MesData.MesCCL);
	MW(WORD_STRONG:= MesBlock1_Temp[1][ 45], SIGNED:=FALSE, FIX:=0 , SIZE:=1, VAR_OUT:=MesDataExd.MesData.MesDCL);
	MW(WORD_STRONG:= MesBlock1_Temp[1][ 46], SIGNED:=TRUE, FIX:=3 , SIZE:=1, VAR_OUT:=MesDataExd.MesData.MesPdc);
	MesDataExd.MesData.MesID_CmdStop_PCS:=MesBlock1_Temp[1][47];
	//MW(WORD_STRONG:= MesBlock1_Temp[1][ 1], SIGNED:=TRUE, FIX:=0 , SIZE:=1, VAR_OUT:=);

	// Block 2 
	MesDataExd.MesData.MesNbRackTot:=MesBlock1_Temp[2][1];
	MesDataExd.MesData.MesNbRackConnected:=MesBlock1_Temp[2][2];
	MW(WORD_STRONG:= MesBlock1_Temp[2][ 3], SIGNED:=TRUE, FIX:=0 , SIZE:=1, VAR_OUT:=MesDataExd.MesData.MesTempMax_Module);
	MesDataExd.MesData.MesIDRack_TempMax_Module:=MesBlock1_Temp[2][4];
	MesDataExd.MesData.MesIDModule_TempMax_Module:=MesBlock1_Temp[2][5];
	MW(WORD_STRONG:= MesBlock1_Temp[2][ 6], SIGNED:=TRUE, FIX:=0 , SIZE:=1, VAR_OUT:=MesDataExd.MesData.MesTempMin_Module);
	MesDataExd.MesData.MesIDRack_TempMin_Module:=MesBlock1_Temp[2][7];
	MesDataExd.MesData.MesIDModule_TempMin_Module:=MesBlock1_Temp[2][8];
	MW(WORD_STRONG:= MesBlock1_Temp[2][ 9], SIGNED:=TRUE, FIX:=0 , SIZE:=1, VAR_OUT:=MesDataExd.MesData.MesTemp_Module);
	//MW(WORD_STRONG:= MesBlock1_Temp[2][ 1], SIGNED:=FALSE, FIX:=0 , SIZE:=1, VAR_OUT:=);
	//MW(WORD_STRONG:= MesBlock1_Temp[2][ 1], SIGNED:=FALSE, FIX:=0 , SIZE:=1, VAR_OUT:=);
	//MW(WORD_STRONG:= MesBlock1_Temp[2][ 1], SIGNED:=FALSE, FIX:=0 , SIZE:=1, VAR_OUT:=);
	//MW(WORD_STRONG:= MesBlock1_Temp[2][ 1], SIGNED:=FALSE, FIX:=0 , SIZE:=1, VAR_OUT:=);
	//MW(WORD_STRONG:= MesBlock1_Temp[2][ 1], SIGNED:=FALSE, FIX:=0 , SIZE:=1, VAR_OUT:=);
	MW(WORD_STRONG:= MesBlock1_Temp[2][ 15], SIGNED:=TRUE, FIX:=1 , SIZE:=1, VAR_OUT:=MesDataExd.MesData.MesImax_Rack);
	MesDataExd.MesData.MesIDRack_Imax_Rack:=MesBlock1_Temp[2][16];
	MW(WORD_STRONG:= MesBlock1_Temp[2][ 17], SIGNED:=TRUE, FIX:=1 , SIZE:=1, VAR_OUT:=MesDataExd.MesData.MesImin_Rack);
	MesDataExd.MesData.MesIDRack_Imin_Rack:=MesBlock1_Temp[2][18];
	MW(WORD_STRONG:= MesBlock1_Temp[2][ 19], SIGNED:=TRUE, FIX:=1 , SIZE:=1, VAR_OUT:=MesDataExd.MesData.MesIdc_Rack);
	MesDataExd.MesData.MesNbCellbalancing:=MesBlock1_Temp[2][20];

	// Block 3 
	MesDataExd.MesNbSubBMS:=MesBlock1_Temp[3][1];
	MW(WORD_STRONG:= MesBlock1_Temp[3][ 2], SIGNED:=FALSE, FIX:=0 , SIZE:=1, VAR_OUT:=MesDataExd.MesEToFullCharge);
	MW(WORD_STRONG:= MesBlock1_Temp[3][ 3], SIGNED:=FALSE, FIX:=0 , SIZE:=1, VAR_OUT:=MesDataExd.MesData.MesEconnected);
	MW(WORD_STRONG:= MesBlock1_Temp[3][ 4], SIGNED:=TRUE, FIX:=2 , SIZE:=1, VAR_OUT:=MesDataExd.MesP_Aux);
	MW(WORD_STRONG:= MesBlock1_Temp[3][ 5], SIGNED:=FALSE, FIX:=2 , SIZE:=1, VAR_OUT:=MesDataExd.MesS_Aux);
	MW(WORD_STRONG:= MesBlock1_Temp[3][ 6], SIGNED:=TRUE, FIX:=2 , SIZE:=1, VAR_OUT:=MesDataExd.MesQ_Aux);
	MW(WORD_STRONG:= MesBlock1_Temp[3][ 7], Word_WEAK:= MesBlock1_Temp[3][8], SIGNED:=FALSE, FIX:=3 , SIZE:=2, VAR_OUT:=MesDataExd.MesEreact_Aux);
	MW(WORD_STRONG:= MesBlock1_Temp[3][ 9], Word_WEAK:= MesBlock1_Temp[3][10], SIGNED:=FALSE, FIX:=3 , SIZE:=2, VAR_OUT:=MesDataExd.MesEact_Aux);
	MW(WORD_STRONG:= MesBlock1_Temp[3][ 11], Word_WEAK:= MesBlock1_Temp[3][12], SIGNED:=FALSE, FIX:=3 , SIZE:=2, VAR_OUT:=MesDataExd.MesEapp_Aux);
	MW(WORD_STRONG:= MesBlock1_Temp[3][ 20], SIGNED:=FALSE, FIX:=1 , SIZE:=1, VAR_OUT:=MesDataExd.MesSoC_Uncertainty);
	MW(WORD_STRONG:= MesBlock1_Temp[3][ 21], SIGNED:=FALSE, FIX:=0 , SIZE:=1, VAR_OUT:=MesDataExd.MesSoEMin);
	MW(WORD_STRONG:= MesBlock1_Temp[3][ 22], SIGNED:=FALSE, FIX:=0 , SIZE:=1, VAR_OUT:=MesDataExd.MesSoEMax);


	// Loop over containers 
	FOR KK:=1 TO CstNbBAT_ESS_G DO 

		ModbusReadBMS[KK]
		(
			pDestAddr 		:= ADR(MesBlockBMS_Temp[KK]),		sIPAddr 		:= ParamIpAddress,			tTimeout 		:= ParamTimeout,
			nTcpPort 		:= ParamTcpPort,				nQuantity 		:= CalBSSModelQty,				nMBAddr 		:= CalRegisterBSSModel,				
			cbLength 		:= SIZEOF(MesBlockBMS_Temp[KK]),	nUnitID 		:= ParamUnitID,				ClockRead 		:= Clockread AND  MesDataExd.MesData.MesCP_Read,
			Reset 			:= IN_CmdReset
		);		
	
		
		
		MW(WORD_STRONG:= MesBlockBMS_Temp[KK][ 1], SIGNED:=FALSE, FIX:=0 , SIZE:=1, VAR_OUT:=MesDataExd.SubBMS[KK].MesEToFullCharge);
		MW(WORD_STRONG:= MesBlockBMS_Temp[KK][ 2], SIGNED:=FALSE, FIX:=0 , SIZE:=1, VAR_OUT:=MesDataExd.SubBMS[KK].MesEconnected);
		MW(WORD_STRONG:= MesBlockBMS_Temp[KK][ 3], SIGNED:=TRUE, FIX:=0 , SIZE:=1, VAR_OUT:=MesDataExd.SubBMS[KK].HVAC.MesTemp_Outside);
		MW(WORD_STRONG:= MesBlockBMS_Temp[KK][ 4], SIGNED:=TRUE, FIX:= , SIZE:=1, VAR_OUT:=MesDataExd.SubBMS[KK].HVAC.MesTemp_Room);
		MW(WORD_STRONG:= MesBlockBMS_Temp[KK][ 5], SIGNED:=FALSE, FIX:= , SIZE:=1, VAR_OUT:=MesDataExd.SubBMS[KK].HVAC.MesHygro_Amb);
		//MW(WORD_STRONG:= MesBlockBMS_Temp[KK][ 1], SIGNED:=FALSE, FIX:= , SIZE:=1, VAR_OUT:=);
		//MW(WORD_STRONG:= MesBlockBMS_Temp[KK][ 1], SIGNED:=FALSE, FIX:= , SIZE:=1, VAR_OUT:=);
		MW(WORD_STRONG:= MesBlockBMS_Temp[KK][ 8], SIGNED:=FALSE, FIX:= , SIZE:=1, VAR_OUT:=MesDataExd.SubBMS[KK].MesU_Aux);
		MW(WORD_STRONG:= MesBlockBMS_Temp[KK][ 9], SIGNED:=FALSE, FIX:= , SIZE:=1, VAR_OUT:=MesDataExd.SubBMS[KK].MesFreq_Aux);
		MW(WORD_STRONG:= MesBlockBMS_Temp[KK][ 10], SIGNED:=FALSE, FIX:=3 , SIZE:=1, VAR_OUT:=MesDataExd.SubBMS[KK].MesP_Aux);
		MW(WORD_STRONG:= MesBlockBMS_Temp[KK][ 11], SIGNED:=FALSE, FIX:=3 , SIZE:=1, VAR_OUT:=MesDataExd.SubBMS[KK].MesS_Aux);
		MW(WORD_STRONG:= MesBlockBMS_Temp[KK][ 12], SIGNED:=FALSE, FIX:=3 , SIZE:=1, VAR_OUT:=MesDataExd.SubBMS[KK].MesQ_Aux);
		MW(WORD_STRONG:= MesBlockBMS_Temp[KK][ 13], Word_WEAK:= MesBlockBMS_Temp[KK][14], SIGNED:=FALSE, FIX:=3 , SIZE:=2, VAR_OUT:=MesDataExd.SubBMS[KK].MesEreact_Aux);
		MW(WORD_STRONG:= MesBlockBMS_Temp[KK][ 15], Word_WEAK:= MesBlockBMS_Temp[KK][16], SIGNED:=FALSE, FIX:=3 , SIZE:=2, VAR_OUT:=MesDataExd.SubBMS[KK].MesEact_Aux);
		MW(WORD_STRONG:= MesBlockBMS_Temp[KK][ 17], Word_WEAK:= MesBlockBMS_Temp[KK][18], SIGNED:=FALSE, FIX:=3 , SIZE:=2, VAR_OUT:=MesDataExd.SubBMS[KK].MesEapp_Aux);
		MW_U(WORD_STRONG:= MesBlockBMS_Temp[KK][ 19], Word_WEAK:= MesBlockBMS_Temp[KK][20], VAR_OUT:=MesDataExd.SubBMS[KK].HVAC.MesIDState);
		MW_U(WORD_STRONG:= MesBlockBMS_Temp[KK][ 21], Word_WEAK:= MesBlockBMS_Temp[KK][22], VAR_OUT:=MesDataExd.SubBMS[KK].MesIDAlarm);
		MW_U(WORD_STRONG:= MesBlockBMS_Temp[KK][ 23], Word_WEAK:= MesBlockBMS_Temp[KK][24], VAR_OUT:=MesDataExd.SubBMS[KK].MesIDAlarm2);

	
	END_FOR 
	
	

END_IF
// RACKS 

// READ TCU DATA 
CTU_ClockRead(CU:=ClockRead , PV:= REAL_TO_WORD(ParamNbRacks/(ParamNbReadAtOnce))+1 ) ; 
CTU_ClockRead(RESET:= CTU_ClockRead.Q ) ; 
LL:= (CTU_ClockRead.CV)  ; // At every Clock Read , we read 10 new racks We reset once all trackers have been read.  


TON_ClockRead(IN:= ClockRead , PT:= ParamClockReadRack_Delay  ) ; // Allow to leave 200ms between the system data read and the racks reading . 

//RACK STRING ( 804)

FOR KK:= 1 TO CstNbRack_BAT_G DO 
		ModbusReadrack[KK]
			(
			pDestAddr 		:= ADR(MesBlockRack_Temp[KK]),		
			sIPAddr 		:= ParamIpAddress,			
			tTimeout 		:= ParamTimeout,
			nTcpPort 		:= ParamTcpPort,				
			nQuantity 		:= 32,				
			nMBAddr 		:= CalRegisterBatModel +26 + 32 *(KK-1) ,				
			cbLength 		:= SIZEOF(MesBlockRack_Temp[KK]),	
			nUnitID 		:= 2,				
			ClockRead 		:= TON_ClockRead.Q AND MesDataExd.MesData.MesCP_Read,
			Reset 			:= IN_CmdReset_L,					
			ModbusReadAlarm => MesModbusReadAlarmRack[KK],	
			ErrorId 		=> MesModbusReadAlarmIDRack[KK]
		);


	// MW 
	
	MesDataExd.RACK[KK].MesData.MesNbModuleTot:=MesBlockRack_Temp[KK][1];
	MW_U(WORD_STRONG:= MesBlockRack_Temp[KK][ 2], Word_WEAK:= MesBlockRack_Temp[KK][3], VAR_OUT:=MesDataExd.RACK[KK].MesData.MesIDState);
	MesDataExd.RACK[KK].MesData.MesID_ConnectFail:=MesBlockRack_Temp[KK][4];
	MW(WORD_STRONG:= MesBlockRack_Temp[KK][ 5], SIGNED:=FALSE, FIX:=1 , SIZE:=1, VAR_OUT:=MesDataExd.RACK[KK].MesData.MesSoC);
	MW(WORD_STRONG:= MesBlockRack_Temp[KK][ 6], SIGNED:=FALSE, FIX:=0 , SIZE:=1, VAR_OUT:=MesDataExd.RACK[KK].MesData.MesSoH);
	MW(WORD_STRONG:= MesBlockRack_Temp[KK][ 7], SIGNED:=TRUE, FIX:=1 , SIZE:=1, VAR_OUT:=MesDataExd.RACK[KK].MesData.MesIdc);
	MW(WORD_STRONG:= MesBlockRack_Temp[KK][ 8], SIGNED:=FALSE, FIX:=3 , SIZE:=1, VAR_OUT:=MesDataExd.RACK[KK].MesData.MesUdcMax_Cell);
	MesDataExd.RACK[KK].MesData.MesIDModule_UdcMax_Cell:=MesBlockRack_Temp[KK][9];
	MW(WORD_STRONG:= MesBlockRack_Temp[KK][ 10], SIGNED:=FALSE, FIX:=3 , SIZE:=1, VAR_OUT:=MesDataExd.RACK[KK].MesData.MesUdcMin_Cell);
	MesDataExd.RACK[KK].MesData.MesIDModule_UdcMin_Cell:=MesBlockRack_Temp[KK][11];
	MW(WORD_STRONG:= MesBlockRack_Temp[KK][ 12], SIGNED:=FALSE, FIX:=3 , SIZE:=1, VAR_OUT:=MesDataExd.RACK[KK].MesData.MesUdc_Cell);
	MW(WORD_STRONG:= MesBlockRack_Temp[KK][ 13], SIGNED:=TRUE, FIX:=0 , SIZE:=1, VAR_OUT:=MesDataExd.RACK[KK].MesData.MesTempMax_Module);
	MesDataExd.RACK[KK].MesData.MesIDModule_TempMax_Module:=MesBlockRack_Temp[KK][14];
	MW(WORD_STRONG:= MesBlockRack_Temp[KK][ 15], SIGNED:=TRUE, FIX:=0 , SIZE:=1, VAR_OUT:=MesDataExd.RACK[KK].MesData.MesTempMin_Module);
	MesDataExd.RACK[KK].MesData.MesIDModule_TempMin_Module:=MesBlockRack_Temp[KK][16];
	MW(WORD_STRONG:= MesBlockRack_Temp[KK][ 17], SIGNED:=TRUE, FIX:=0 , SIZE:=1, VAR_OUT:=MesDataExd.RACK[KK].MesData.MesTemp_Module);
	MesDataExd.RACK[KK].MesData.MesID_Disable:=MesBlockRack_Temp[KK][18];
	MW_U(WORD_STRONG:= MesBlockRack_Temp[KK][ 19], Word_WEAK:= MesBlockRack_Temp[KK][20], VAR_OUT:=MesDataExd.RACK[KK].MesData.MesIDState_DCSwitch);
	MW_U(WORD_STRONG:= MesBlockRack_Temp[KK][ 21], Word_WEAK:= MesBlockRack_Temp[KK][22], VAR_OUT:=MesDataExd.RACK[KK].MesData.MesIDAlarm);
	//MW(WORD_STRONG:= MesBlock2_Temp[KK][ 1], SIGNED:=FALSE, FIX:=0 , SIZE:=1, VAR_OUT:=);
	MW_U(WORD_STRONG:= MesBlockRack_Temp[KK][ 25], Word_WEAK:= MesBlockRack_Temp[KK][26], VAR_OUT:=MesDataExd.RACK[KK].MesData.MesIDAlarm_Vendor1);
	MW_U(WORD_STRONG:= MesBlockRack_Temp[KK][ 27], Word_WEAK:= MesBlockRack_Temp[KK][28], VAR_OUT:=MesDataExd.RACK[KK].MesData.MesIDAlarm_Vendor2);
	//MW(WORD_STRONG:= MesBlock2_Temp[KK][ 29], SIGNED:=FALSE, FIX:=0 , SIZE:=1, VAR_OUT:=);
	//MW(WORD_STRONG:= MesBlock2_Temp[KK][ 30], SIGNED:=FALSE, FIX:=0 , SIZE:=1, VAR_OUT:=);
	MW(WORD_STRONG:= MesBlockRack_Temp[KK][ 31], SIGNED:=FALSE, FIX:=1 , SIZE:=1, VAR_OUT:=MesDataExd.RACK[KK].MesData.MesSoC_Uncertainty);


END_FOR





(*FOR KK:= 1 TO ParamNbReadAtOnce DO 
	
	CalRackNb := LL*ParamNbReadAtOnce+KK; 	
	IF CalRackNb > ParamNbRacks THEN 
		EXIT ; 
	END_IF	
	
	IF MesDataExd.MesData.MesCP_Read THEN
		ModbusReadrack[(ParamNbModule+1)*(KK-1)+1]
			(
			pDestAddr 		:= ADR(MesBlock2_Temp[(ParamNbModule+1)*(KK-1)+1]),		
			sIPAddr 		:= ParamIpAddress,			
			tTimeout 		:= ParamTimeout,
			nTcpPort 		:= ParamTcpPort,				
			nQuantity 		:= AX_Qty[2],				
			nMBAddr 		:= AX_Addr[2] + (CalRackNb-1)*360,				
			cbLength 		:= SIZEOF(MesBlock2_Temp[(ParamNbModule+1)*(KK-1)+1]),	
			nUnitID 		:= 2,				
			ClockRead 		:= TON_ClockRead.Q AND MesDataExd.MesData.MesCP_Read,
			Reset 			:= IN_CmdReset_L,					
			ModbusReadAlarm => MesModbusReadAlarm2[(ParamNbModule+1)*(KK-1)+1],	
			ErrorId 		=> MesModbusReadAlarmID2[(ParamNbModule+1)*(KK-1)+1]
		);
	

	// DATA
		IF ModbusReadrack[(ParamNbModule+1)*(KK-1)+1].OUT_Completed THEN 
//		MesDataExd.MesData.AX_Rack[CalRackNb].ParamNbStrings:=MesBlock2_Temp[(ParamNbRackString+1)*(KK-1)+1][0];
		
		
		
		END_IF
	END_IF
	
	*)
	
	
	// RACK MODULE ( 805)
		FOR KK:= 1 TO CstNbModule_Rack_G DO 
	
		ModbusReadmodule[KK]
			(
			pDestAddr 		:= ADR(MesBlockRack_Temp[KK]),		
			sIPAddr 		:= ParamIpAddress,			
			tTimeout 		:= ParamTimeout,
			nTcpPort 		:= ParamTcpPort,				
			nQuantity 		:= 32,				
			nMBAddr 		:= CalRegisterBatModel +26 + 32 *(KK-1) ,				
			cbLength 		:= SIZEOF(MesBlockRack_Temp[KK]),	
			nUnitID 		:= 2,				
			ClockRead 		:= TON_ClockRead.Q AND MesDataExd.MesData.MesCP_Read,
			Reset 			:= IN_CmdReset_L,					
			ModbusReadAlarm => MesModbusReadAlarmRack[KK],	
			ErrorId 		=> MesModbusReadAlarmIDRack[KK]
		);		
		
		
		
		
		
		
		
		
				
			MesDataExd.RACK[KK].Module[JJ].MesNbCell:=MesBlockModule_Temp[KK][1];
			MW(WORD_STRONG:= MesBlockModule_Temp[KK][ 1], SIGNED:=FALSE, FIX:=0 , SIZE:=1, VAR_OUT:=MesDataExd.RACK[KK].Module[JJ].MesSoC);
			MW(WORD_STRONG:= MesBlockModule_Temp[KK][ 1], SIGNED:=FALSE, FIX:=0 , SIZE:=1, VAR_OUT:=MesDataExd.RACK[KK].Module[JJ].MesSoH);
			MW(WORD_STRONG:= MesBlockModule_Temp[KK][ 4], SIGNED:=FALSE, FIX:=3 , SIZE:=1, VAR_OUT:=MesDataExd.RACK[KK].Module[JJ].MesUdcMax_Cell);
			MW(WORD_STRONG:= MesBlockModule_Temp[KK][ 1], SIGNED:=FALSE, FIX:=0 , SIZE:=1, VAR_OUT:=MesDataExd.RACK[KK].Module[JJ].MesIDCell_UdcMax_Cell);
			MW(WORD_STRONG:= MesBlockModule_Temp[KK][ 6], SIGNED:=FALSE, FIX:=3 , SIZE:=1, VAR_OUT:=MesDataExd.RACK[KK].Module[JJ].MesUdcMin_Cell);
			MesDataExd.RACK[KK].Module[JJ].MesIDCell_UdcMin_Cell:=MesBlockModule_Temp[KK][7];
			MW(WORD_STRONG:= MesBlockModule_Temp[KK][ 8], SIGNED:=FALSE, FIX:=3 , SIZE:=1, VAR_OUT:=MesDataExd.RACK[KK].Module[JJ].MesUdc_Cell);
			MW(WORD_STRONG:= MesBlockModule_Temp[KK][ 9], SIGNED:=TRUE, FIX:=0 , SIZE:=1, VAR_OUT:=MesDataExd.RACK[KK].Module[JJ].MesTempMax_Cell);
			MW(WORD_STRONG:= MesBlockModule_Temp[KK][ 1], SIGNED:=FALSE, FIX:=0 , SIZE:=1, VAR_OUT:=MesDataExd.RACK[KK].Module[JJ].MesIDCell_TempMax_Cell);
			MW(WORD_STRONG:= MesBlockModule_Temp[KK][ 11], SIGNED:=TRUE, FIX:=0 , SIZE:=1, VAR_OUT:=MesDataExd.RACK[KK].Module[JJ].MesTempMin_Cell);
			MW(WORD_STRONG:= MesBlockModule_Temp[KK][ 1], SIGNED:=FALSE, FIX:=0 , SIZE:=1, VAR_OUT:=MesDataExd.RACK[KK].Module[JJ].MesIDCell_TempMin_Cell);
			MW(WORD_STRONG:= MesBlockModule_Temp[KK][ 13], SIGNED:=TRUE, FIX:=0 , SIZE:=1, VAR_OUT:=MesDataExd.RACK[KK].Module[JJ].MesTemp_Cell);
			
					
		
		
		
	
	
		
		
	
	
		END_FOR 
	
	FOR JJ:= 1 TO ParamNbModule DO 
		IF MesDataExd.MesData.MesCP_Read THEN	
			ModbusReadrack[(ParamNbModule+1)*(KK-1)+JJ+1]
				(
				pDestAddr 		:= ADR(MesBlockRack_Temp[(ParamNbModule+1)*(KK-1)+JJ+1]),		
				sIPAddr 		:= ParamIpAddress,			
				tTimeout 		:= ParamTimeout,
				nTcpPort 		:= ParamTcpPort,				
				nQuantity 		:= AX_Qty[3],				
				nMBAddr 		:= AX_Addr[2] + (CalRackNb-1)*360 + JJ*120,				
				cbLength 		:= SIZEOF(MesBlockRack_Temp[(ParamNbModule+1)*(KK-1)+JJ+1]),	
				nUnitID 		:= 3,				
				ClockRead 		:= TON_ClockRead.Q AND MesDataExd.MesData.MesCP_Read,
				Reset 			:= IN_CmdReset_L,					
				ModbusReadAlarm => MesModbusReadAlarmRack[(ParamNbModule+1)*(KK-1)+JJ+1],	
				ErrorId 		=> MesModbusReadAlarmIDRack[(ParamNbModule+1)*(KK-1)+JJ+1]
			);

		//DATA
			IF ModbusReadrack[(ParamNbModule+1)*(KK-1)+JJ+1].OUT_Completed THEN 
//			MesDataExd.MesData.AX_RACK[CalrackNb].AX_RACKSTRING[JJ].MesMode:=MesBlock2_Temp[(ParamNbRackString+1)*(KK-1)+JJ+1][0];
	
			END_IF
		END_IF


	END_FOR 

//END_FOR


SUPER^.M_Read();
END_METHOD

METHOD M_StartStop
//////////////////
//  Start or stop BBMS via CAN bus   
/////////////////

VAR 
	// Method local variables (reinitialized at each cycle) 
		KK			: INT;

		CP_Start	: BOOL;
		CI_RPM		: BOOL;
		CI_BIR		: BOOL;
		CI_IDC1		: BOOL;
		CI_IDC2		: BOOL ; 
		CI_BS		: BOOL;
		CI_BST		: BOOL;
		CI_RSR		: BOOL;
		CI_FCR		: BOOL;
		CI_ESTP		: BOOL;
END_VAR

SUPER^.M_StartStop();
END_METHOD

METHOD M_StateManager
//////////////////
// Detect which is the state of the PCS system . 
/////////////////

VAR 
	// Method local variables (reinitialized at each cycle) 

	
END_VAR
MesDataExd.MesData.MesState  		:= 0 ; 
(*
IF MesDataExd.MesSystemMode.8 THEN
	CalState.2 := 1;
ELSIF MesDataExd.MesSystemMode.7 THEN
	CalState.1 := 1;
ELSIF MesDataExd.MesSystemMode.6 THEN
	CalState.0 := 1;
END_IF

*)
	
SUPER^.M_StateManager() ;
END_METHOD

METHOD M_Write
VAR_INPUT
END_VAR
VAR
	InputAddr: WORD;
	RTCWord: ARRAY[1..6] OF BYTE;
	TriggerRTC: BOOL;
END_VAR
(*
Trig_CmdCloseDC(CLK := IN_CmdCloseDC);
Trig_CmdOpenDC(CLK := IN_CmdOpenDC);
Trig_CmdReset(CLK := IN_CmdReset_L);

IF Trig_CmdCloseDC.Q THEN
	IN_CmdCloseDC := FALSE;
	AX_Cmd[1] := 1;
END_IF
IF Trig_CmdOpenDC.Q THEN
	IN_CmdOpenDC := FALSE;
	AX_Cmd[1] := 2;
END_IF


IF Trig_CmdReset.Q AND NOT AX_ESS[ParamEssNum].AX_PCS[1].MesState>1 THEN			// lacth the fault date of events. WE HAVE TO CHECK FIRST THE FAULT BEFORE DOING IT// The Reset shall be disabled if the PCS is started/ 
	IN_CmdReset_L := FALSE;
	AX_Cmd[2] := 1;
END_IF

Trig_Watchdog(CLK := CalLocalTimeStruct.wSecond MOD 5 = 0 );	// watchdog every 5 seconds . 
IF Trig_Watchdog.Q THEN
	AX_Cmd[3] := CalLocalTimeStruct.wSecond;
END_IF


IF AX_ESS[ParamEssNum].AX_PCS[1].MesDataExd.MesData.MesState.1 THEN 
	AX_Cmd[4] :=  1 ; // PCS Off 
ELSIF AX_ESS[ParamEssNum].AX_PCS[1].MesDataExd.MesData.MesState.2 THEN
	AX_Cmd[4] :=  2 ; // PCS Standy 
ELSE
	AX_Cmd[4] :=  3 ;	// PCS started 
END_IF


AX_ModbusWrite[1]
(
	InputWord	:= AX_Cmd[1],
	sIPAddr 	:= ParamIpAddress,
	tTimeout 	:= ParamTimeout,
	nTCPport 	:= ParamTcpPort,
	nMBAddr 	:= 48,
	nUnitID 	:= ParamUnitID,
	WriteCmd 	:= Trig_CmdCloseDC.Q OR Trig_CmdOpenDC.Q AND MesDataExd.MesData.MesCP_Write ,
);




AX_ModbusWrite[2]
(
	InputWord	:= AX_Cmd[2],
	sIPAddr 	:= ParamIpAddress,
	tTimeout 	:= ParamTimeout,
	nTCPport 	:= ParamTcpPort,
	nMBAddr 	:= 18,
	nUnitID 	:= ParamUnitID,
	WriteCmd 	:= Trig_CmdReset.Q AND MesDataExd.MesData.MesCP_Write,
);

AX_ModbusWrite[3]	// Wa&tchdog / Heartbit 
(
	InputWord	:= AX_Cmd[3],
	sIPAddr 	:= ParamIpAddress,
	tTimeout 	:= ParamTimeout,
	nTCPport 	:= ParamTcpPort,
	nMBAddr 	:= 17,
	nUnitID 	:= ParamUnitID,
	WriteCmd 	:= Trig_Watchdog.Q AND MesDataExd.MesData.MesCP_Write,
);


// PCS State 
AX_ModbusWrite[4]	// PCS State
(
	InputWord	:= AX_Cmd[4],
	sIPAddr 	:= ParamIpAddress,
	tTimeout 	:= ParamTimeout,
	nTCPport 	:= ParamTcpPort,
	nMBAddr 	:= 49,
	nUnitID 	:= ParamUnitID,
	WriteCmd 	:= ClockWrite AND MesDataExd.MesData.MesCP_Write,
);




// Write Datetime to BMS to keep same date . 
RTCWord[1] := WORD_TO_BYTE(2000 - CalLocalTimeStruct.wYear) ; 
RTCWord[2] :=  WORD_TO_BYTE(CalLocalTimeStruct.wMonth); 
RTCWord[3] := WORD_TO_BYTE(CalLocalTimeStruct.wDay); 
RTCWord[4] := WORD_TO_BYTE(CalLocalTimeStruct.wHour); 
RTCWord[5] := WORD_TO_BYTE(CalLocalTimeStruct.wMinute); 
RTCWord[6] := WORD_TO_BYTE(CalLocalTimeStruct.wSecond); 

TriggerRTC := CalLocalTimeStruct.wHour = 5 AND CalLocalTimeStruct.wMinute = 0 AND CalLocalTimeStruct.wSecond = 0 ; // Write dat once a day

A1_ModbusWriteRTC	// 
(   
	cbLength :=  SIZEOF(RTCWord ) ,
	pSrcAddr	:= ADR(RTCWord) , 
	nQuantity	:= 3 ,
	sIPAddr 	:= ParamIpAddress,
	tTimeout 	:= ParamTimeout,
	nTCPport 	:= ParamTcpPort,
	nMBAddr 	:= 0,
	nUnitID 	:= ParamUnitID,
	WriteCmd 	:=  (TriggerRTC) AND MesDataExd.MesData.MesCP_Write,
	Reset				:= CmdClearFault_G, 
);


	
SUPER^.M_Write();

*)
END_METHOD

END_FUNCTION_BLOCK

// ---- 01_Equipement_Library/Batteries/FUN_AlarmManagement_STR.TcPOU
PROGRAM FUN_AlarmManagement_STR
VAR
END_VAR

METHOD M_AlarmManagement : BOOL
VAR_INPUT
	Alarm1 		: WORD;
	Alarm2 		: WORD;
	Alarm3 		: WORD;
	Alarm4 		: WORD;
	Protection1 : WORD;
	Protection2 : WORD;
	Protection3 : WORD;
	Protection4 : WORD;
END_VAR
VAR
	FB_AlarmCodeManager 		: FB_AlarmCodeManager ; 
END_VAR
VAR_OUTPUT
	MesProtection1 	: WORD;
	MesProtection2 	: WORD;
	MesAlarm1 		: WORD;
	MesAlarm2 		: WORD;
END_VAR
	FB_AlarmCodeManager(
		bAlarm1			:= Protection4.0,			// BMS Protection4 module_pcb_ut
		bAlarm2			:= Protection4.1,			// BMS Protection4 module_pcb_ot
		bAlarm3			:= Protection4.2,       	// BMS Protection4 dcsw_count_fail
		bAlarm4			:= Protection4.8,       	// BMS Protection4 fuse_or_dcsw_sensing_fail
		bAlarm5			:= Protection3.8,       	// BMS Protection3_dcsw1_sensing_fail
		bAlarm6			:= Protection3.9,       	// BMS Protection3_dcsw2_sensing_fail
		bAlarm7			:= Protection3.10,      	// BMS Protection3_dcsw1_fail
		bAlarm8			:= Protection3.11,      	// BMS Protection3_dcsw2_fail
		bAlarm9			:= Protection3.12,      	// BMS Protection3_fan_fail_Option
		bAlarm10		:= Protection3.13,      	// BMS Protection3_additional_protection_fail
		bAlarm11		:= Protection3.14,      	// BMS Protection3_cell_chg_operation_limit
		bAlarm12		:= Protection3.15,      	// BMS Protection3_cell_dchg_operation_limit
		bAlarm13		:= Protection1.0,       	// BMS_Protection1_module_UT
		bAlarm14		:= Protection1.1,       	// BMS_Protection1_module_OT
		bAlarm15		:= Protection1.2,       	// BMS_Protection1_module_UV
	wAlarmCode		=> MesProtection1);
	
	FB_AlarmCodeManager(
		bAlarm1			:= Protection1.3,			// BMS_Protection1_module_OV
		bAlarm2			:= Protection1.4,			// BMS_Protection1_module_V_imb
		bAlarm3			:= Protection1.5,			// BMS_Protection1_module_T_imb
		bAlarm4			:= Protection1.6,    		// BMS_Protection1_R_M_comm_fail
		bAlarm5			:= Protection1.7,    		// BMS_Protection1_R_S_comm_fail
		bAlarm6			:= Protection1.8,    		// BMS_Protection1_rack_ChgOC
		bAlarm7			:= Protection1.9,    		// BMS_Protection1_rack_DchgOC
		bAlarm8			:= Protection1.10,   		// BMS_Protection1_rack_UV
		bAlarm9			:= Protection1.11,   		// BMS_Protection1_rack_OV
		bAlarm10		:= Protection1.12,    		// BMS_Protection1_rack_V_sensing_diff
		bAlarm11		:= Protection1.13,    		// BMS_Protection1_rack_I_senser_fail
		bAlarm12		:= Protection1.14,    		// BMS_Protection1_rack_fuse_fail_Option
		bAlarm13		:= Protection1.15,    		// BMS_Protection1_permanent_uv
		bAlarm14		:= FALSE, // 
		bAlarm15		:= False, // 
	wAlarmCode		=> MesProtection2);

		FB_AlarmCodeManager(
		bAlarm1			:= Alarm4.0,			// BMS Alarm4 module_pcb_ut
		bAlarm2			:= Alarm4.1,			// BMS Alarm4 module_pcb_ot
		bAlarm3			:= Alarm4.2,       		// BMS Alarm4 dcsw_count_fail
		bAlarm4			:= Alarm4.8,       		// BMS Alarm4 fuse_or_dcsw_sensing_fail
		bAlarm5			:= Alarm3.8,       		// BMS Alarm3 dcsw1_sensing_fail
		bAlarm6			:= Alarm3.9,       		// BMS Alarm3 dcsw2_sensing_fail
		bAlarm7			:= Alarm3.10,      		// BMS Alarm3 dcsw1_fail
		bAlarm8			:= Alarm3.11,      		// BMS Alarm3 dcsw2_fail
		bAlarm9			:= Alarm3.12,      		// BMS Alarm3 fan_fail_Option
		bAlarm10		:= Alarm3.13,      		// BMS Alarm3 additional_protection_fail
		bAlarm11		:= Alarm3.14,      		// BMS Alarm3 cell_chg_operation_limit
		bAlarm12		:= Alarm3.15,      		// BMS Alarm3 cell_dchg_operation_limit
		bAlarm13		:= Alarm1.0,       		// BMS Alarm1 module_UT
		bAlarm14		:= Alarm1.1,       		// BMS Alarm1 module_OT
		bAlarm15		:= Alarm1.2,       		// BMS Alarm1 module_UV
	wAlarmCode		=> MesAlarm1);
	
	FB_AlarmCodeManager(
		bAlarm1			:= Alarm1.4,			// BMS Alarm1_module_OV
		bAlarm2			:= Alarm1.4,			// BMS Alarm1_module_V_imb
		bAlarm3			:= Alarm1.5,			// BMS Alarm1_module_T_imb
		bAlarm4			:= Alarm1.6,    		// BMS Alarm1_R_M_comm_fail
		bAlarm5			:= Alarm1.7,    		// BMS Alarm1_R_S_comm_fail
		bAlarm6			:= Alarm1.8,    		// BMS Alarm1_rack_ChgOC
		bAlarm7			:= Alarm1.9,    		// BMS Alarm1_rack_DchgOC
		bAlarm8			:= Alarm1.10,   		// BMS Alarm1_rack_UV
		bAlarm9			:= Alarm1.11,   		// BMS Alarm1_rack_OV
		bAlarm10		:= Alarm1.12,    		// BMS Alarm1_rack_V_sensing_diff
		bAlarm11		:= Alarm1.13,    		// BMS Alarm1_rack_I_senser_fail
		bAlarm12		:= Alarm1.14,    		// BMS Alarm1_rack_fuse_fail_Option
		bAlarm13		:= Alarm1.15,    		// BMS Alarm1_permanent_uv
		bAlarm14		:= FALSE, // 
		bAlarm15		:= False, // 
	wAlarmCode		=> MesAlarm2);
END_METHOD

END_PROGRAM

// ---- 01_Equipement_Library/Datalogger/FB_Datalogger_Base.TcPOU
FUNCTION_BLOCK FB_Datalogger_Base

VAR_INPUT PERSISTENT
	ParamTcpPort				: UINT	:=	502;		 (* (NA) Modbus TCP port*)
	ParamIPAddress				: STRING;				 (* (NA) Config: IP Adress *)
	ParamUnitID					: BYTE;					 (* (NA) Modbus Unit ID *)
	ParamClockRead 				: TIME 	:= TIME#2S; 	 (* (Time) Read Modbus frequency  	*)
	
	bInit						: BOOL  := TRUE; 		 // (NA) Initialisation 
END_VAR

VAR_INPUT           	
	IN_CmdToggleRead			: BOOL;
	IN_CmdToggleWrite			: BOOL;
	IN_CmdReset_L				: BOOL;
END_VAR             	
      	
VAR                 	
//INPUT
	ClockRead					: BOOL;							// (NA) Modbus reading Clock
    TP1							: TP ; 							// (NA) Tempo to define Modbus Reading Frequency 
	
	Trig_Cmd_Read				: R_Trig;
	Trig_Cmd_Write              : R_Trig;
	
//  MesDataExd.MesData.                    : Datalogger;
END_VAR

VAR PERSISTENT

END_VAR

METHOD M_AlarmManagement
//////////////////
// Generates object alarms and manages resets. 
//////////////////

VAR 
	// Method local variables (reinitialized at each cycle) 
	FB_AlarmCodeManager		: FB_AlarmCodeManager ;  
END_VAR
END_METHOD

METHOD M_CP

VAR 
	// Method local variables (reinitialized at each cycle) 
	
END_VAR
END_METHOD

METHOD M_Execute : BOOL
VAR_INPUT
END_VAR
	
	TP1(IN:=NOT TP1.Q , PT:= ParamClockRead );
	ClockRead 	:= TP1.Q;
	
	M_CP();
		
	M_Read();
	
	M_Write();
	
	M_AlarmManagement();
END_METHOD

METHOD M_Read : BOOL
VAR_INPUT
END_VAR

VAR
	MW					: FB_MergeWordsToFloat;
END_VAR
END_METHOD

METHOD M_Write : BOOL
VAR
		CmdbyCom	: WORD;
		
END_VAR
END_METHOD

END_FUNCTION_BLOCK

// ---- 01_Equipement_Library/Datalogger/FB_Datalogger_IOWIT.TcPOU
FUNCTION_BLOCK FB_Datalogger_IOWIT EXTENDS FB_Datalogger_Base

VAR_INPUT PERSISTENT
	{attribute 'OPC.UA.DA' := '1'} 
	ParamTcpPort			: UINT   := 502;					(* Modbus TCP port															*)
	{attribute 'OPC.UA.DA' := '1'}                          	
	ParamIPAddress			: STRING;				 			(* (NA)Config: IP Adress of WIT                                             *)
	{attribute 'OPC.UA.DA' := '1'} 	                        	
	ParamUnitID 			: BYTE:=1; 							(* (NA)   SMA Modbus Unit ID.                                               *)
	                                                        	
	ParamTempoComAlarm		: TIME 		:= T#30S ; 				(* (s) Config : Tempo to detect LOC Alarm                                   *)
	ParamTimeOutCurtail     : TIME 		:= T#45S ;				(* (s) Config : Tempo to curtail power at set value before Timeout warning  *)
	ParamClockReadTime 		: TIME 		:= TIME#2S;	  			(* (Time) Read Modbus Frequency .                                           *)
	ParamClockWriteTime 	: TIME 		:= TIME#2S; 	  		(* (Time) Write Modbus Frequency .                                          *)
 	ParamTimeout			: TIME  	:= T#5S ;		  		(* (Time) Timeout for modbus reading                                        *)
		                                                    
	ParamID					: UINT :=1; 						(* ID of the datalogger . Corresponding to PTR ID .                         *)
	
END_VAR

VAR_INPUT 
	// Parameters of the Object (instance specific) 
	IN_CmdToggleRead			: BOOL ;
		
	IN_CmdReset_L				: BOOL ;						// (NA) External Reset Command
	                                                    		
	MbAddrDI	: WORD; 										// Adresse IP Requête Digital Inputs
	MbAddrAI	: ARRAY[1.. 8] OF WORD; 						// Adresses IP Requête Analogic Inputs 
	
	MesDataExd AT %Q*			      	: Datalogger_IOWIT ; 	// (NA) [P,H,B] INV  Data Structure 

	
	
	
END_VAR

VAR
		
	// M_READ VARIABLES//
	
	
	FB_ModbusReadDI	        : FB_ModbusReadCoils;   	 		// FB for Modbus Reading Digital Values
	FB_ModbusReadAI			: FB_ModbusRead;			 		// FB for Modbus Reading Analogic Values (Adresses on 1010X-1019X range)
	
	DI_List : ARRAY[1..27] OF BOOL;
	AI_List : ARRAY[1..18] OF WORD;
	TempAIList : ARRAY[1..2] OF WORD;
		
		
	// M_ALARMMNGMT VARIABLES //
	TON_ComAlarm				: TON ; 						// Tempo before deteting loss of communication. 
	TON_ComWarning				: TON ; 						// Tempo before detecting loss of communication.                                                	
                                 		    	        		
	MesComWarning				: BOOL ; 						// (NA) [P,H]  True if bad communication
                                                        		
	                                                    		
	//M_EXECUTE VARIABLES //                            		
	TP1							: TP ; 	 						// (NA) Tempo to define Modbus Reading Frequency 
	Trig_Cmd_Read: R_TRIG;	                            	
	                                                    	
	ClockRead		AT %Q*		: BOOL	;						// (NA) Modbus reading Clock
    
    
	bInit						: BOOL;
	
	
END_VAR

METHOD M_AlarmManagement
//////////////////
// Manages IntelliGen Alarms
/////////////////

VAR 
	// Method local variables (reinitialized at each cycle) 
	FB_AlarmCodeManager : FB_AlarmCodeManager ; 
	KK				: BYTE;		// For Loop 
	bComError		: BOOL := TRUE;
	bComWarning 	: BOOL;
	AC_CB_OPEN		: BOOL;
END_VAR

// ALARM CODE //
	FB_AlarmCodeManager(
		bAlarm1			:= MesDataExd.MesData.Transfo.MesDataExd.MesData.MesAlarmTemp , 		// A1_Transfo : Temperature alarm
		bAlarm2			:= MesDataExd.MesData.FSS.MesAlarmFire , 					// FSS : Security Fire Detection                                         
		bAlarm3			:= MesDataExd.MesData.Transfo.MesDataExd.MesData.MesAlarmGas ,			// A1_Transfo : Transfo Gaz Discharge                                      
		bAlarm4			:= MesDataExd.MesData.Transfo.MesDataExd.MesData.MesAlarmOilLevel ,	// A1_Transfo : Transfo Pressure 	                                           
		bAlarm5			:= MesDataExd.MesData.MS.MesAlarmState , 					// A1_MS : Security Motion Sensor                                         
		bAlarm6			:= MesDataExd.MesData.DS.MesAlarmState ,					// A1_DS : Security Door Contact                                           
		bAlarm7			:= MesDataExd.MesData.WS.MesSVS_Signal1,					// A1_WS : Security Video Signal 1                                          
		bAlarm8			:= MesDataExd.MesData.WS.MesSVS_Signal2,					// A1_WS : Security Video Signal 2            
		bAlarm9			:= MesDataExd.MesData.WS.MesSVS_Signal3,					// A1_WS : Security Video Signal 3            
		bAlarm10		:= MesDataExd.MesData.CB_Transfo.MesAlarmState, 			// CB_Transfo : Alarm State                                         
		bAlarm11		:= MesDataExd.MesData.CB_INV[1].MesAlarmState, 				// CB_INV_1 : Alarm State                                         
		bAlarm12		:= MesDataExd.MesData.CB_INV[2].MesAlarmState, 				// CB_INV_2 : Alarm State                                         
		bAlarm13		:=FALSE, //                                          
		bAlarm14		:=FALSE, //                                          
		bAlarm15		:=FALSE , 			// 			                                 
		wAlarmCode		=>MesDataExd.MesData.MesAlarmCode);                            

// WARNING CODE //
	FB_AlarmCodeManager(
 		bAlarm1			:= MesDataExd.MesData.Transfo.MesDataExd.MesData.MesWarningTemp,		//	A1_Transfo : Transfo Temp Warning 		
		bAlarm2			:=FALSE, //
		bAlarm3			:=FALSE, //
		bAlarm4			:=FALSE, //                                 
		bAlarm5			:=FALSE, //                          	
		bAlarm6			:=FALSE, //                                   
		bAlarm7			:=FALSE, //                                   
		bAlarm8			:=FALSE, //                                   
		bAlarm9			:=FALSE, //                                   
		bAlarm10		:=FALSE, //                                   
		bAlarm11		:=FALSE, //                                   
		bAlarm12		:=FALSE, //                                   
		bAlarm13		:=FALSE, //                                   
		bAlarm14		:=FALSE, //                                   
		bAlarm15		:=FALSE, //                                   
		wAlarmCode		=>MesDataExd.MesData.MesWarningCode);

// EVENT CODE //
	FB_AlarmCodeManager(
 		bAlarm1			:= MesDataExd.MesData.MesInvReturnContact1, // Inverter Return Contact 1		
		bAlarm2			:= MesDataExd.MesData.MesInvReturnContact2, // Inverter Return Contact 2
		bAlarm3			:=FALSE, //
		bAlarm4			:=FALSE, //                                 
		bAlarm5			:=FALSE, //                          	
		bAlarm6			:=FALSE, //                                   
		bAlarm7			:=FALSE, //                                   
		bAlarm8			:=FALSE, //                                   
		bAlarm9			:=FALSE, //                                   
		bAlarm10		:=FALSE, //                                   
		bAlarm11		:=FALSE, //                                   
		bAlarm12		:=FALSE, //                                   
		bAlarm13		:=FALSE, //                                   
		bAlarm14		:=FALSE, //                                   
		bAlarm15		:=FALSE, //                                   
		wAlarmCode		=>MesDataExd.MesData.MesWarningCode);
END_METHOD

METHOD M_CP
//////////////////
//  Emulator
/////////////////

VAR 
	// Method local variables (reinitialized at each cycle) 
	

END_VAR


SUPER^.M_CP() ; 




Trig_Cmd_Read(CLK:=IN_CmdToggleRead);
Trig_Cmd_Write(CLK:=IN_CmdToggleWrite);
	
IF Trig_Cmd_Read.Q THEN
	IN_CmdToggleRead := FALSE;
	MesDataExd.MesData.MesCP_Read := NOT MesDataExd.MesData.MesCP_Read;
END_IF


IF Trig_Cmd_Write.Q THEN
	IN_CmdToggleWrite := FALSE;
	MesDataExd.MesData.MesCP_Write := NOT MesDataExd.MesData.MesCP_Write;
END_IF
END_METHOD

METHOD M_Execute
//////////////////
//  Method Calls 
/////////////////

VAR 
	// Method local variables (reinitialized at each cycle) 

END_VAR
M_CP() ; 
M_Read() ; 
M_AlarmManagement() ;
END_METHOD

{attribute 'object_name' := 'M_Read'}
METHOD M_Read
//////////
// Read Method for SMA : Modbus reading
//////////
VAR
	// Method local variables (reinitialized at each cycle) 
	//MW					: FB_MergeWordsToFloat;
	//MW_1				: FB_WordsToDint64BE;
	

	MW					: FB_MergeWordsToDint;
	i 					: INT;
	
	MesInv2SSM6SwitchGear: INT;
	KK: INT;
END_VAR

// CP-Read / Write 


IF MesDataExd.MesData.MesCP_Read  THEN		 
	
	// Digital Inputs Modbus Requests 
	
	FB_ModbusReadDI(pDestAddr := ADR(DI_List),
					sIPAddr := ParamIPAddress,
					tTimeout := ParamTimeout,
					nTcpPort := 502,
					nQuantity := 28,
					nMBAddr := MbAddrDI,
					cbLength := SIZEOF(DI_List),
					nUnitID := 1,
					ClockRead := MesDataExd.MesData.MesCP_Read AND ClockRead,
					Reset := CmdClearFault_G OR IN_CmdReset_L);
					
	FOR i := 1 TO 8 DO
		FB_ModbusReadAI(pDestAddr := ADR(TempAIList),
					sIPAddr := ParamIPAddress,
					tTimeout := ParamTimeout,
					nTcpPort := 502,
					nQuantity := 2,
					nMBAddr := MbAddrAI[i],
					cbLength := SIZEOF(TempAIList),
					nUnitID := 1,
					ClockRead := MesDataExd.MesData.MesCP_Read AND ClockRead,
					Reset := CmdClearFault_G OR IN_CmdReset_L);
					
		AI_List[2*i-1] := TempAIList[1];
		AI_List[2*i] := TempAIList[2];
	END_FOR	
	
	//  MesDataExd.MesData.Filling Digital Input			
	
	MesDataExd.MesData.MesInvReturnContact1	:=	DI_List[1]; 	
	MesDataExd.MesData.MesInvReturnContact2	:=	DI_List[2]; 
		
	MesDataExd.MesData.Transfo.MesDataExd.MesData.MesAlarmGas 			:= DI_List[3];
	MesDataExd.MesData.Transfo.MesDataExd.MesData.MesAlarmOilLevel 		:= DI_List[4];
	MesDataExd.MesData.Transfo.MesDataExd.MesData.MesWarningTemp 		:= DI_List[5];
	MesDataExd.MesData.Transfo.MesDataExd.MesData.MesAlarmTemp        	:= DI_List[6];
	
	MesDataExd.MesData.CB_Transfo.MesAlarmState	:=	DI_List[7];	// NO ? 
	MesDataExd.MesData.FSS.MesAlarmFire      		:=  DI_List[8];
	 
	MesDataExd.MesData.CB_INV[1].MesAlarmState 	:=	DI_List[9]; 
	MesDataExd.MesData.CB_INV[2].MesAlarmState  	:= 	DI_List[10];
	 
	MesDataExd.MesData.MS.MesAlarmState 	:=	DI_List[11];
	MesDataExd.MesData.DS.MesAlarmState 	:=  DI_List[12];			// MesSecurityDoorContact
	MesDataExd.MesData.WS.MesSVS_Signal1 	:=  DI_List[13];
		
	 FOR KK:= 1 TO CstNbSTR_G DO 
	 	AX_PTR[ParamID].AX_INV[1].MesDataExd.MesData.Fuse_DC[KK].MesAlarmState 	:=	DI_List[14+(KK-1)];		// MesInv1SSM1SwitchGear
	 END_FOR
	  FOR KK:= 1 TO CstNbSTR_G DO 
	 	AX_PTR[ParamID].AX_INV[2].MesDataExd.MesData.Fuse_DC[KK].MesAlarmState 	:=	DI_List[20+(KK-1)];		// MesInv1SSM1SwitchGear
	 END_FOR
	 
	
	MesDataExd.MesData.WS.MesSVS_Signal2	:=	DI_List[26];
	MesDataExd.MesData.WS.MesSVS_Signal3 :=  DI_List[27];
	 
	 
	 
	 (*
	MesDataExd.MesData.MesInvReturnContact1	:=	DI_List[1]; 	
	MesDataExd.MesData.MesInvReturnContact2	:=	DI_List[2]; 
		
	MesDataExd.MesData.MesTransfoGazDischarge		:= DI_List[3];
	MesDataExd.MesData.MesTransfoPressure		   	:= DI_List[4];
	MesDataExd.MesData.MesTransfoTempWarning		:= DI_List[5];
	MesDataExd.MesData.MesTransfoTempTrig        	:= DI_List[6];
	
	MesDataExd.MesData.MesHVAuxSwitchGearTransfo	:=	DI_List[7];
	MesDataExd.MesData.MesSecurityFireDetect     	:=  DI_List[8];
	 
	MesDataExd.MesData.MesHVAuxSwitchGearInv1	:=	DI_List[9]; 
	MesDataExd.MesData.MesHVAuxSwitchGearInv2  := 	DI_List[10];
	 
	MesDataExd.MesData.MesSecurityMotionSensor	:=	DI_List[11];
	MesDataExd.MesData.MesSecurityDoorContact	:=  DI_List[12];
	MesDataExd.MesData.A1_WS.MesSVS_Signal1 :=  DI_List[13];
		
	MesDataExd.MesData.MesInv1SSM1SwitchGear	:=	DI_List[14];
	MesDataExd.MesData.MesInv1SSM2SwitchGear	:=	DI_List[15];
	MesDataExd.MesData.MesInv1SSM3SwitchGear   :=  DI_List[16];
	MesDataExd.MesData.MesInv1SSM4SwitchGear	:=  DI_List[17];
	MesDataExd.MesData.MesInv1SSM5SwitchGear   :=  DI_List[18];
	MesDataExd.MesData.MesInv1SSM6SwitchGear	:=  DI_List[19];
	MesDataExd.MesData.MesInv2SSM1SwitchGear   :=  DI_List[20];
	MesDataExd.MesData.MesInv2SSM2SwitchGear   :=  DI_List[21];
	MesDataExd.MesData.MesInv2SSM3SwitchGear   :=  DI_List[22];
	MesDataExd.MesData.MesInv2SSM4SwitchGear   :=  DI_List[23];
	MesDataExd.MesData.MesInv2SSM5SwitchGear   :=  DI_List[24];
	MesDataExd.MesData.MesInv2SSM6SwitchGear   :=  DI_List[25];
	*)
	
	
	//  MesDataExd.MesData.Filling Analogic Input
	
	
	MW(WORD_STRONG :=  AI_List[1],	WORD_WEAK := AI_List[2], SIZE := 1, FIX := 0, SIGNED := 0, VAR_OUT	:= MesDataExd.MesData.MesTransfoLocalTemp);
	MW(WORD_STRONG :=  AI_List[3],	WORD_WEAK := AI_List[4], SIZE := 1, FIX := 0, SIGNED := 0, VAR_OUT	:= MesDataExd.MesData.WS.MesTempMod1);
	MW(WORD_STRONG :=  AI_List[5],	WORD_WEAK := AI_List[6], SIZE := 1, FIX := 0, SIGNED := 0, VAR_OUT	:= MesDataExd.MesData.WS.MesTempMod2);
	MW(WORD_STRONG :=  AI_List[7],	WORD_WEAK := AI_List[8], SIZE := 1, FIX := 0, SIGNED := 0, VAR_OUT	:= MesDataExd.MesData.WS.MesTempExt);
	MW(WORD_STRONG :=  AI_List[9],	WORD_WEAK := AI_List[10], SIZE := 1, FIX := 0, SIGNED := 0, VAR_OUT	:= MesDataExd.MesData.WS.MesWindSpd);		
	MW(WORD_STRONG :=  AI_List[11],	WORD_WEAK := AI_List[12], SIZE := 1, FIX := 0, SIGNED := 0, VAR_OUT	:= MesDataExd.MesData.WS.MesGHI_Left);	  
	MW(WORD_STRONG :=  AI_List[13],	WORD_WEAK := AI_List[14], SIZE := 1, FIX := 0, SIGNED := 0, VAR_OUT	:= MesDataExd.MesData.WS.MesGHI_Middle);	
	MW(WORD_STRONG :=  AI_List[15],	WORD_WEAK := AI_List[16], SIZE := 1, FIX := 0, SIGNED := 0, VAR_OUT	:= MesDataExd.MesData.WS.MesGHI_Right);	 
	
END_IF
END_METHOD

END_FUNCTION_BLOCK

// ---- 01_Equipement_Library/Datalogger/FB_Datalogger_SchSkid.TcPOU
FUNCTION_BLOCK FB_Datalogger_SchSkid EXTENDS FB_Datalogger_Base
 

VAR_INPUT PERSISTENT
	ParamID_PTR					: BYTE; 				 						(* (NA) ID of the datalogger. Corresponding to PTR ID *)
	ParamWriteTimeout			: TIME  	:= T#5S ;		  					(* (Time) Timeout for modbus reading*)
END_VAR

       	
VAR_INPUT           	
	// I/O Inputs 
	MesDataExd  AT %Q*		: Datalogger_SchSkid;
END_VAR             	
      	
VAR                 	


	CmdbyCom 		AT %Q*		: WORD;
	
//INPUT Modbus
	FB_ModbusRead	          	: ARRAY[1..2] OF FB_ModbusRead; 	            // (NA) FB for Modbus Reading
	FB_COMWrite					: FB_ModbusWrite;
	MesBlock1_Temp				: ARRAY [1..19] OF WORD ; 
	MesBlock2_Temp 				: ARRAY [1..26] OF WORD ; 
	
	ModbusInputBoolAlarms		: BOOL;
	ModbusInputBoolAlarmId		: UDINT;
	ModbusInputAnaAlarms		: BOOL;
	ModbusInputAnaAlarmId		: UDINT;
	TEMP_4_20					: ARRAY [1..13] OF REAL;

//OUTPUT Modbus
	MesModbusCmdByComAlarm 		: BOOL;
	MesModbusCmdByComCodeId		: UDINT;
	Front_Montant				: R_Trig;
	RS_Open						: RS;
	RS_Close					: RS;
	
END_VAR

METHOD M_AlarmManagement
//////////////////
// Generates object alarms and manages resets. 
//////////////////

VAR 
	// Method local variables (reinitialized at each cycle) 
	FB_AlarmCodeManager		: FB_AlarmCodeManager;  
END_VAR
	
// ALARM CODE //
	FB_AlarmCodeManager(
		bAlarm1				:= MesDataExd.Transfo_Synthesis.MesData.MesAlarmsSynthesis,		// Synthesis : trip of DGPT2 ON G,P,T (from DI_208)
		bAlarm2				:= MesDataExd.Transfo_Synthesis.MesData.MesAlarmTemp,			// Synthesis : alarms temperature (from DI_207) 
		bAlarm3				:= MesDataExd.DS_Synthesis.MesData.MesAlarmState,						// Synthesis : door positions (from DI_209)
		bAlarm4				:= FALSE,														//
		bAlarm5				:= FALSE,														//
		bAlarm6				:= FALSE,														//
		bAlarm7				:= FALSE,														//
		bAlarm8				:= FALSE,														//
		bAlarm9				:= FALSE,														//
		bAlarm10			:= FALSE,														//
		bAlarm11			:= MesDataExd.CB_INV[1].MesData.MesAlarmState, 							// CB_INV_1 : alarm state 
		bAlarm12			:= MesDataExd.CB_INV[2].MesData.MesAlarmState, 							// CB_INV_2 : alarm state 
		bAlarm13			:= FALSE, 														//                                          
		bAlarm14			:= FALSE,														//                                          
		bAlarm15			:= FALSE,														// 		
		wAlarmCode			=>MesDataExd.MesData.MesAlarmCode);										//
			
// WARNING CODE //
	FB_AlarmCodeManager(
		bAlarm1				:= FALSE, 														// 
		bAlarm2				:= FALSE, 														//
		bAlarm3				:= FALSE,														//
		bAlarm4				:= FALSE,														//
		bAlarm5				:= FALSE,														//
		bAlarm6				:= FALSE,														//
		bAlarm7				:= FALSE,														//
		bAlarm8				:= FALSE,														//
		bAlarm9				:= FALSE,														//
		bAlarm10			:= FALSE,														//
		bAlarm11			:= FALSE,														//
		bAlarm12			:= FALSE,														//
		bAlarm13			:= FALSE,														//
		bAlarm14			:= FALSE,														//
		bAlarm15			:= FALSE,														//
		wAlarmCode			=>MesDataExd.MesData.MesWarningCode);										//
		                                                        							
// EVENT CODE //                                                							
                                                                							
	FB_AlarmCodeManager(                                        							
		bAlarm1				:= FALSE,						    							//  
		bAlarm2				:= FALSE, 														//  
		bAlarm3				:= FALSE,														//
		bAlarm4				:= FALSE,														//
		bAlarm5				:= FALSE,														//
		bAlarm6				:= FALSE,														//
		bAlarm7				:= FALSE,														//
		bAlarm8				:= FALSE,														//
		bAlarm9				:= FALSE,														//
		bAlarm10			:= FALSE,														//
		bAlarm11			:= FALSE,														//
		bAlarm12			:= FALSE,														//
		bAlarm13			:= FALSE,														//
		bAlarm14			:= FALSE,														//
		bAlarm15			:= FALSE,														//
		wAlarmCode			=>MesDataExd.MesData.MesEventCode);										//
END_METHOD

METHOD M_CP

VAR 
	// Method local variables (reinitialized at each cycle) 
	
END_VAR


SUPER^.M_CP() ; 




Trig_Cmd_Read(CLK:=IN_CmdToggleRead);
Trig_Cmd_Write(CLK:=IN_CmdToggleWrite);
	
IF Trig_Cmd_Read.Q THEN
	IN_CmdToggleRead := FALSE;
	MesDataExd.MesData.MesCP_Read := NOT MesDataExd.MesData.MesCP_Read;
END_IF


IF Trig_Cmd_Write.Q THEN
	IN_CmdToggleWrite := FALSE;
	MesDataExd.MesData.MesCP_Write := NOT MesDataExd.MesData.MesCP_Write;
END_IF
END_METHOD

METHOD M_Execute : BOOL
VAR_INPUT
END_VAR
IF bInit THEN
	M_Init();
	bInit := FALSE;
ELSIF CmdInit_G THEN 
	bInit:= TRUE ;
END_IF

SUPER^.M_Execute() ;
END_METHOD

METHOD M_Init : BOOL
VAR_INPUT
END_VAR
END_METHOD


METHOD M_Read : BOOL
VAR_INPUT
END_VAR

VAR
	MW					: FB_MergeWordsToFloat;
END_VAR
// CP-Read / Write 


IF MesDataExd.MesData.MesCP_Read  THEN	
//DI MODBUS	
	FB_ModbusRead[1]
		(
			nTCPPort		:= ParamTcpPort,
			ClockRead		:= MesDataExd.MesData.MesCP_Read AND ClockRead, 
			Reset			:= CmdClearFault_G OR IN_CmdReset_L,
			sIPAddr			:= ParamIPAddress ,
			nUnitID			:= 1, 
			tTimeout		:= T#5S,
			nQuantity		:= 19, 
			nMBAddr			:= 300 , 
			cbLength		:= SIZEOF(MesBlock1_Temp), 
			pDestAddr		:= ADR(MesBlock1_Temp), 
			ModbusReadAlarm	=> ModbusInputBoolAlarms, 
			ErrorId			=> ModbusInputBoolAlarmId
		);
//4-20ma MODBUS	
		FB_ModbusRead[2]
		(
			nTCPPort		:= ParamTcpPort,
			ClockRead		:= MesDataExd.MesData.MesCP_Read AND ClockRead, 
			Reset			:= CmdClearFault_G OR IN_CmdReset_L,
			sIPAddr			:= ParamIPAddress ,
			nUnitID			:= 1, 
			tTimeout		:= T#5S,
			nQuantity		:= 26, 
			nMBAddr			:= 400 , 
			cbLength		:= SIZEOF(MesBlock2_Temp), 
			pDestAddr		:= ADR(MesBlock2_Temp), 
			ModbusReadAlarm	=> ModbusInputAnaAlarms, 
			ErrorId			=> ModbusInputAnaAlarmId
		);

	
//DI	
MesDataExd.MesWatchdog_ProtectRelayVIP 						:= WORD_TO_BOOL(MesBlock1_Temp[1]);
MesDataExd.CB_INV[1].MesData.MesAlarmState							:= WORD_TO_BOOL(MesBlock1_Temp[2]);
MesDataExd.CB_INV[2].MesData.MesAlarmState							:= WORD_TO_BOOL(MesBlock1_Temp[3]); 
MesDataExd.MesComutLocal									:= WORD_TO_BOOL(MesBlock1_Temp[4]);
MesDataExd.MesState_MVCB									:= WORD_TO_BOOL(MesBlock1_Temp[5]);
MesDataExd.MesFault_ProtectRelayVIP							:= WORD_TO_BOOL(MesBlock1_Temp[6]);
MesDataExd.Transfo_Synthesis.MesData.MesAlarmTemp			:= WORD_TO_BOOL(MesBlock1_Temp[7]);
MesDataExd.Transfo_Synthesis.MesData.MesAlarmsSynthesis		:= WORD_TO_BOOL(MesBlock1_Temp[8]);
MesDataExd.DS_Synthesis.MesData.MesAlarmState						:= WORD_TO_BOOL(MesBlock1_Temp[9]); 				// TRUE OUVERT
	
	IF 	ParamID_PTR	= 4 THEN
	MesDataExd.CB_INV[1].MesData.MesAlarmState 						:= MesDataExd.CB_INV[2].MesData.MesAlarmState; 				// CB of inverter one is in inverter 2
	END_IF	
	
//4-20ma
	MW( WORD_STRONG:= MesBlock2_Temp[2  ],	WORD_WEAK := MesBlock2_Temp[1  ], VAR_OUT :=Temp_4_20[1] ); 		//
    MW( WORD_STRONG:= MesBlock2_Temp[4  ], 	WORD_WEAK := MesBlock2_Temp[3  ], VAR_OUT :=Temp_4_20[2] ); 		// 
    MW( WORD_STRONG:= MesBlock2_Temp[6  ], 	WORD_WEAK := MesBlock2_Temp[5  ], VAR_OUT :=Temp_4_20[3] ); 		// 
    MW( WORD_STRONG:= MesBlock2_Temp[8  ], 	WORD_WEAK := MesBlock2_Temp[7  ], VAR_OUT :=Temp_4_20[4] ); 		// 
    MW( WORD_STRONG:= MesBlock2_Temp[10 ], 	WORD_WEAK := MesBlock2_Temp[9  ], VAR_OUT :=Temp_4_20[5] );		// 
    MW( WORD_STRONG:= MesBlock2_Temp[12 ], 	WORD_WEAK := MesBlock2_Temp[11 ], VAR_OUT :=Temp_4_20[6] );  
    MW( WORD_STRONG:= MesBlock2_Temp[14 ], 	WORD_WEAK := MesBlock2_Temp[13 ], VAR_OUT :=Temp_4_20[7] );		// Pyrano route PTR1,2,4 / wind speed for PTR3
    MW( WORD_STRONG:= MesBlock2_Temp[16 ], 	WORD_WEAK := MesBlock2_Temp[15 ], VAR_OUT :=Temp_4_20[8] ); 		// Pyrano eau PTR1,2,4 / wind direction for PTR3
    MW( WORD_STRONG:= MesBlock2_Temp[18 ], 	WORD_WEAK := MesBlock2_Temp[17 ], VAR_OUT :=Temp_4_20[9] ); 		// Temp panel
    MW( WORD_STRONG:= MesBlock2_Temp[20 ], 	WORD_WEAK := MesBlock2_Temp[19 ], VAR_OUT :=Temp_4_20[10]); 
    MW( WORD_STRONG:= MesBlock2_Temp[22 ], 	WORD_WEAK := MesBlock2_Temp[21 ], VAR_OUT :=Temp_4_20[11]); 
    //MW( WORD_STRONG_F:= MesBlock2_Temp[24 ], 	WORD_WEAK_F := MesBlock2_Temp[23 ], NUMBER_F := MesDataExd.MesData.MesTemp_TrasfoOil_1  ); // Tp Transfo 1
	//MW( WORD_STRONG_F:= MesBlock2_Temp[26 ], 	WORD_WEAK_F := MesBlock2_Temp[25 ], NUMBER_F := MesDataExd.MesData.MesTemp_TrasfoOil_2  ); // Tp Transfo 2
END_IF
END_METHOD

METHOD M_Write : BOOL
VAR
		
		
END_VAR
IF AX_PTR[ParamID_PTR].A1_MainMVCB_PTR.OUT_CmdClose_IO THEN
	CmdbyCom.0 := 0;
	CmdbyCom.1 := 1;
END_IF
	
IF AX_PTR[ParamID_PTR].A1_MainMVCB_PTR.OUT_CmdOpen_IO THEN
	CmdbyCom.0 := 1;
	CmdbyCom.1 := 0;
END_IF

Front_Montant(CLK:= AX_PTR[ParamID_PTR].A1_MainMVCB_PTR.OUT_CmdClose_IO OR AX_PTR[ParamID_PTR].A1_MainMVCB_PTR.OUT_CmdOpen_IO);
RS_Open(SET:=Front_Montant.Q,Reset1:= NOT MesDataExd.MesState_MVCB OR IN_CmdReset_L );

RS_Close(SET:=Front_Montant.Q,Reset1:=MesDataExd.MesState_MVCB OR IN_CmdReset_L);


FB_COMWrite(
		pSrcAddr 			:= ADR(CmdbyCom) ,
		cbLength			:= SIZEOF(CmdbyCom) , 
		nQuantity 			:= 1,
		Reset				:= CmdClearFault_G OR IN_CmdReset_L, 
		sIPAddr				:= ParamIPAddress , 
		nUnitID				:= 1 , //modif LWN
		nMBAddr				:= 40302 , 
		tTimeout			:= ParamWriteTimeout ,
		WriteCmd			:= (RS_Open.Q1 OR RS_close.Q1) AND MesDataExd.MesData.MesCP_Write, 
		ModbusWriteAlarm	=> MesModbusCmdByComAlarm , 
		ErrorId				=> MesModbusCmdByComCodeId);
END_METHOD

END_FUNCTION_BLOCK

// ---- 01_Equipement_Library/Datalogger/FB_Datalogger_SENECA.TcPOU
FUNCTION_BLOCK FB_Datalogger_SENECA EXTENDS FB_Datalogger_Base
 

VAR_INPUT PERSISTENT
	ParamWriteTimeout			: TIME  	:= T#5S ;		  					(* (Time) Timeout for modbus reading*)
END_VAR

       	
VAR_INPUT           	
	// I/O Inputs 
	MesDataExd				: Datalogger_SENECA;    
END_VAR             	
      	
VAR 
            		
	
//INPUT Modbus
	FB_ModbusRead	          	: ARRAY[1..2] OF FB_ModbusRead; 	            // (NA) FB for Modbus Reading	
	MesBlock1_Temp				: ARRAY [1..8] OF WORD ; 
	
	AlarmModbusInput			: BOOL;
	AlarmID_ModbusInput			: UDINT;
END_VAR

METHOD M_AlarmManagement
//////////////////
// Generates object alarms and manages resets 
//////////////////

VAR 
	// Method local variables (reinitialized at each cycle) 
	FB_AlarmCodeManager		: FB_AlarmCodeManager;  
	Transfo_Synthesis		: INT;
END_VAR
	
// ALARM CODE //
	FB_AlarmCodeManager(
		bAlarm1				:= FALSE,														// 
		bAlarm2				:= FALSE,														// 
		bAlarm3				:= FALSE,														// 
		bAlarm4				:= FALSE,														//
		bAlarm5				:= FALSE,														//
		bAlarm6				:= FALSE,														//
		bAlarm7				:= FALSE,														//
		bAlarm8				:= FALSE,														//
		bAlarm9				:= FALSE,														//
		bAlarm10			:= FALSE,														//
		bAlarm11			:= FALSE, 														// 
		bAlarm12			:= FALSE, 														// 
		bAlarm13			:= FALSE, 														//                                          
		bAlarm14			:= FALSE,														//                                          
		bAlarm15			:= FALSE,														// 		
		wAlarmCode			=>MesDataExd.MesData.MesAlarmCode);										//
			
// WARNING CODE //
	FB_AlarmCodeManager(
		bAlarm1				:= AlarmModbusInput, 											// Error Modbus read of the datalogger data
		bAlarm2				:= FALSE, 														//
		bAlarm3				:= FALSE,														//
		bAlarm4				:= FALSE,														//
		bAlarm5				:= FALSE,														//
		bAlarm6				:= FALSE,														//
		bAlarm7				:= FALSE,														//
		bAlarm8				:= FALSE,														//
		bAlarm9				:= FALSE,														//
		bAlarm10			:= FALSE,														//
		bAlarm11			:= FALSE,														//
		bAlarm12			:= FALSE,														//
		bAlarm13			:= FALSE,														//
		bAlarm14			:= FALSE,														//
		bAlarm15			:= FALSE,														//
		wAlarmCode			=>MesDataExd.MesData.MesWarningCode);										//
		                                                        							
// EVENT CODE //                                                							                                                     							
	FB_AlarmCodeManager(                                        							
		bAlarm1				:= FALSE,						    							//  
		bAlarm2				:= FALSE, 														//  
		bAlarm3				:= FALSE,														//
		bAlarm4				:= FALSE,														//
		bAlarm5				:= FALSE,														//
		bAlarm6				:= FALSE,														//
		bAlarm7				:= FALSE,														//
		bAlarm8				:= FALSE,														//
		bAlarm9				:= FALSE,														//
		bAlarm10			:= FALSE,														//
		bAlarm11			:= FALSE,														//
		bAlarm12			:= FALSE,														//
		bAlarm13			:= FALSE,														//
		bAlarm14			:= FALSE,														//
		bAlarm15			:= FALSE,														//
		wAlarmCode			=>MesDataExd.MesData.MesEventCode);										//
		
MesDataExdMesDataExd		:= MesDataExd.MesData.
END_METHOD

METHOD M_CP

VAR 
	// Method local variables (reinitialized at each cycle) 
	
END_VAR


SUPER^.M_CP() ; 




Trig_Cmd_Read(CLK:=IN_CmdToggleRead);
Trig_Cmd_Write(CLK:=IN_CmdToggleWrite);
	
IF Trig_Cmd_Read.Q THEN
	IN_CmdToggleRead := FALSE;
	MesDataExd.MesData.MesCP_Read := NOT MesDataExd.MesData.MesCP_Read;
END_IF


IF Trig_Cmd_Write.Q THEN
	IN_CmdToggleWrite := FALSE;
	MesDataExd.MesData.MesCP_Write := NOT MesDataExd.MesData.MesCP_Write;
END_IF
END_METHOD

METHOD M_Execute : BOOL
VAR_INPUT
END_VAR
IF bInit THEN
	M_Init();
	bInit := FALSE;
ELSIF CmdInit_G THEN 
	bInit:= TRUE ;
END_IF

SUPER^.M_Execute() ;
END_METHOD

METHOD M_Init : BOOL
VAR_INPUT
END_VAR
END_METHOD


METHOD M_Read : BOOL
VAR_INPUT
END_VAR

VAR
	MW					: FB_MergeWordsToFloat;
END_VAR
// CP-Read / Write 


IF MesDataExd.MesData.MesCP_Read  THEN	
// MODBUS Read	
	FB_ModbusRead[1]
		(
			nTCPPort		:= ParamTcpPort,
			ClockRead		:= MesDataExd.MesData.MesCP_Read AND ClockRead, 
			Reset			:= CmdClearFault_G OR IN_CmdReset_L,
			sIPAddr			:= ParamIPAddress ,
			nUnitID			:= 1, 
			tTimeout		:= ParamWriteTimeout,
			nQuantity		:= 4, 
			nMBAddr			:= 40005, 
			cbLength		:= SIZEOF(MesBlock1_Temp), 
			pDestAddr		:= ADR(MesBlock1_Temp), 
			ModbusReadAlarm	=> AlarmModbusInput, 
			ErrorId			=> AlarmID_ModbusInput
		);
	
// Wind Data : Float AB CD	
	MW( WORD_STRONG:= MesBlock1_Temp[1  ],	WORD_WEAK := MesBlock1_Temp[2  ], VAR_OUT := MesDataExd.MesData.MesWindSp);		
	MW( WORD_STRONG:= MesBlock1_Temp[3  ],	WORD_WEAK := MesBlock1_Temp[4  ], VAR_OUT := MesDataExd.MesData.MesWindDir);
END_IF
END_METHOD

METHOD M_Write : BOOL
VAR
		
		
END_VAR
END_METHOD

END_FUNCTION_BLOCK

// ---- 01_Equipement_Library/GRID/FB_GRID_Base.TcPOU
FUNCTION_BLOCK FB_GRID_Base 
//////////////////
// Grid Operator interface. Base FB.
//////////////////
VAR_INPUT PERSISTENT
	// Parameters of the Object (instance specific) 
	
END_VAR

VAR_INPUT
	// I/O Inputs 
		MesConnectOrderIO			: BOOL ; 					// (NA) 
		MesDisconnectOrderIO 		: BOOL ; 					// (NA) 	
		
END_VAR

VAR_OUTPUT
	//Child objects
	
END_VAR
VAR
	//M_ALARMMANAGEMENT VARIABLES//                                                    								
//	MesDataExd				: GRID ;                   								
		
	//M_INIT VARIABLES //
		bInit						: BOOL:= TRUE ; 			// (NA) Initialize object parameters at first cycle 
		
	// M_EXECUTE VARIABLES //
	
   		MesCP_Read					: BOOL := TRUE;	(* Read function enable *)
		

                      	
END_VAR

METHOD M_AlarmManagement
//////////////////
// Digiware measurement tool alarm and warning management
/////////////////

VAR 
	
END_VAR
END_METHOD

METHOD M_CP

VAR 
	// Method local variables (reinitialized at each cycle) 
	
END_VAR
END_METHOD

METHOD M_Evaluate
//////////////////
//  Read Modbus Variable for PCS. 
/////////////////
VAR 
	// Method local variables (reinitialized at each cycle) 
	
END_VAR
END_METHOD

METHOD M_Execute
//////////////////
//  Method Calls 
/////////////////
VAR 
	// Method local variables (reinitialized at each cycle) 

END_VAR

// PERMANENT CONDITIONS //
	M_CP() ; 
	
// METHODS CALLS //
	IF bInit THEN
		M_Init() ; 
		bInit					:= FALSE ; 
	ELSIF CmdInit_G THEN 
		bInit:= TRUE ;
		
	END_IF

	M_Evaluate() ; 
	M_AlarmManagement();
END_METHOD

METHOD M_Init
VAR 

END_VAR
END_METHOD

END_FUNCTION_BLOCK

// ---- 01_Equipement_Library/GRID/FB_GRID_Enedis.TcPOU
FUNCTION_BLOCK FB_GRID_Enedis EXTENDS FB_GRID_Base
//////////////////
// Grid Operator interface. Base FB
//////////////////
VAR_INPUT PERSISTENT
	// Parameters of the Object (instance specific) 
		{attribute 'OPC.UA.DA' := '1'} 
		ParamRseAvailable						: BOOL:=TRUE;		(* (NA) GRID with RSE option*)
		{attribute 'OPC.UA.DA' := '1'} 
		ParamTaAvailable						: BOOL:=TRUE;		(* (NA) GRID with Teleaction option*)
		{attribute 'OPC.UA.DA' := '1'} 
		ParamP0Available						: BOOL:=TRUE; 		(* (NA) GRID with P regulation option*)
		{attribute 'OPC.UA.DA' := '1'} 
		ParamQ0Available						: BOOL:=TRUE; 		(* (NA) GRID with Q regulation option*)
		{attribute 'OPC.UA.DA' := '1'} 
		ParamU0Available						: BOOL:=TRUE; 		(* (NA) GRID with U regulation option*)
		{attribute 'OPC.UA.DA' := '1'} 
		ParamPmaxPark							: REAL;				(* (kW) Contractual maximal power plant active power*)
		{attribute 'OPC.UA.DA' := '1'} 
		ParamPMin								: REAL;				(* (kW)   Contractual minimal power plant active power*)
		{attribute 'OPC.UA.DA' := '1'} 
		ParamQMax								: REAL;				(* (Kvar) Contractual maximal power plant reactive power*)
		{attribute 'OPC.UA.DA' := '1'} 
		ParamQMin								: REAL; 			(* (Kvar) Contractual maximal power plant reactive power*)
		{attribute 'OPC.UA.DA' := '1'} 
		ParamUMax								: REAL;				(* (Kvar) Contractual maximal power plant reactive power*)
		{attribute 'OPC.UA.DA' := '1'} 
		ParamUMin								: REAL; 			(* (Kvar) Contractual maximal power plant reactive power*)
		
		ParamTONFiltering						: TIME:=T#200MS; 	(* (ms) Minimum tempo filter before command validation (noise filtering)*)
		
		MesDataExd								: GRID_Enedis;    
		
END_VAR


